  MoveL 1331 to (-194.97, 429.6, -4.48) mm, rotated rx -180 ry 0 rz -11.91 deg; joints [13.946, -29.664, 81.646, -88.075, 90.999, 141.138]
  MoveL 1332 to (-195.21, 429.6, -4.47) mm, rotated rx -180 ry 0 rz -11.91 deg; joints [13.938, -29.668, 81.653, -88.081, 90.994, 141.141]
  MoveL 1333 to (-195.45, 429.58, -4.47) mm, rotated rx -180 ry 0 rz -11.91 deg; joints [13.931, -29.672, 81.662, -88.087, 90.989, 141.146]
  MoveL 1334 to (-195.69, 429.55, -4.48) mm, rotated rx -180 ry 0 rz -11.91 deg; joints [13.923, -29.676, 81.673, -88.093, 90.984, 141.152]
  MoveL 1335 to (-195.93, 429.49, -4.47) mm, rotated rx -180 ry 0 rz -11.91 deg; joints [13.916, -29.682, 81.686, -88.098, 90.979, 141.159]
  MoveL 1336 to (-196.18, 429.42, -4.47) mm, rotated rx -180 ry 0 rz -11.91 deg; joints [13.909, -29.689, 81.701, -88.104, 90.974, 141.167]
  MoveL 1337 to (-196.42, 429.32, -4.47) mm, rotated rx -180 ry 0 rz -11.91 deg; joints [13.902, -29.698, 81.719, -88.109, 90.97, 141.176]
  MoveL 1338 to (-196.6, 429.23, -4.48) mm, rotated rx -180 ry 0 rz -11.91 deg; joints [13.896, -29.704, 81.734, -88.113, 90.966, 141.184]
  MoveL 1339 to (-196.78, 429.13, -4.47) mm, rotated rx -180 ry 0 rz -11.91 deg; joints [13.891, -29.712, 81.751, -88.117, 90.963, 141.193]
  MoveL 1340 to (-196.95, 429, -4.48) mm, rotated rx -180 ry 0 rz -11.91 deg; joints [13.887, -29.721, 81.769, -88.121, 90.96, 141.203]
  MoveL 1341 to (-197.13, 428.87, -4.48) mm, rotated rx -180 ry 0 rz -11.91 deg; joints [13.882, -29.73, 81.79, -88.124, 90.956, 141.214]
  MoveL 1342 to (-197.37, 428.65, -4.47) mm, rotated rx -180 ry 0 rz -11.91 deg; joints [13.876, -29.744, 81.82, -88.128, 90.952, 141.231]
  MoveL 1343 to (-197.56, 428.44, -4.47) mm, rotated rx -180 ry 0 rz -11.91 deg; joints [13.872, -29.758, 81.85, -88.132, 90.949, 141.246]
  MoveL 1344 to (-197.72, 428.22, -4.48) mm, rotated rx 180 ry 0 rz -11.91 deg; joints [13.868, -29.771, 81.878, -88.134, 90.946, 141.262]
  MoveL 1345 to (-197.85, 428.01, -4.48) mm, rotated rx 180 ry 0 rz -11.91 deg; joints [13.865, -29.783, 81.906, -88.136, 90.944, 141.277]
  MoveL 1346 to (-197.98, 427.77, -4.47) mm, rotated rx -180 ry 0 rz -11.91 deg; joints [13.863, -29.797, 81.937, -88.137, 90.942, 141.293]
  MoveL 1347 to (-198.08, 427.53, -4.48) mm, rotated rx -180 ry 0 rz -11.91 deg; joints [13.862, -29.811, 81.966, -88.138, 90.941, 141.309]
  MoveL 1348 to (-198.16, 427.29, -4.48) mm, rotated rx -180 ry 0 rz -11.91 deg; joints [13.861, -29.825, 81.996, -88.138, 90.94, 141.325]
  MoveL 1349 to (-198.21, 427.04, -4.48) mm, rotated rx -180 ry 0 rz -11.91 deg; joints [13.861, -29.838, 82.024, -88.138, 90.94, 141.34]
  MoveL 1350 to (-198.25, 426.8, -4.48) mm, rotated rx -180 ry 0 rz -11.91 deg; joints [13.862, -29.851, 82.053, -88.137, 90.94, 141.356]
  MoveL 1351 to (-198.27, 426.56, -4.48) mm, rotated rx 180 ry 0 rz -11.91 deg; joints [13.864, -29.864, 82.08, -88.136, 90.94, 141.37]
  MoveL 1352 to (-198.27, 426.08, -4.48) mm, rotated rx 180 ry 0 rz -11.91 deg; joints [13.867, -29.889, 82.134, -88.133, 90.941, 141.4]
  MoveL 1353 to (-198.27, 425.59, -4.48) mm, rotated rx -180 ry 0 rz -11.91 deg; joints [13.871, -29.914, 82.188, -88.129, 90.943, 141.429]
  MoveL 1354 to (-198.25, 425.35, -4.47) mm, rotated rx -180 ry 0 rz -11.91 deg; joints [13.874, -29.926, 82.215, -88.127, 90.944, 141.443]
  MoveL 1355 to (-198.22, 425.11, -4.47) mm, rotated rx -180 ry 0 rz -11.91 deg; joints [13.877, -29.938, 82.241, -88.124, 90.945, 141.457]
  MoveL 1356 to (-198.16, 424.87, -4.48) mm, rotated rx -180 ry 0 rz -11.91 deg; joints [13.881, -29.95, 82.266, -88.121, 90.947, 141.471]
  MoveL 1357 to (-198.09, 424.63, -4.48) mm, rotated rx -180 ry 0 rz -11.91 deg; joints [13.885, -29.961, 82.291, -88.117, 90.949, 141.484]
  MoveL 1358 to (-197.99, 424.39, -4.48) mm, rotated rx -180 ry 0 rz -11.91 deg; joints [13.89, -29.972, 82.315, -88.113, 90.952, 141.498]
  MoveL 1359 to (-197.87, 424.15, -4.47) mm, rotated rx -180 ry 0 rz -11.91 deg; joints [13.896, -29.983, 82.339, -88.108, 90.955, 141.51]
  MoveL 1360 to (-197.73, 423.93, -4.48) mm, rotated rx 180 ry 0 rz -11.91 deg; joints [13.902, -29.993, 82.36, -88.103, 90.959, 141.522]
  MoveL 1361 to (-197.57, 423.71, -4.47) mm, rotated rx -180 ry 0 rz -11.91 deg; joints [13.91, -30.002, 82.38, -88.097, 90.963, 141.532]
  MoveL 1362 to (-197.38, 423.49, -4.48) mm, rotated rx 180 ry 0 rz -11.91 deg; joints [13.918, -30.011, 82.399, -88.09, 90.967, 141.543]
  MoveL 1363 to (-197.14, 423.27, -4.47) mm, rotated rx -180 ry 0 rz -11.91 deg; joints [13.927, -30.019, 82.417, -88.083, 90.973, 141.553]
  MoveL 1364 to (-196.96, 423.13, -4.47) mm, rotated rx -180 ry 0 rz -11.91 deg; joints [13.934, -30.025, 82.428, -88.077, 90.977, 141.558]
  MoveL 1365 to (-196.78, 423, -4.48) mm, rotated rx 180 ry 0 rz -11.91 deg; joints [13.941, -30.029, 82.436, -88.071, 90.981, 141.563]
  MoveL 1366 to (-196.6, 422.9, -4.48) mm, rotated rx -180 ry 0 rz -11.91 deg; joints [13.948, -30.032, 82.443, -88.066, 90.985, 141.567]
  MoveL 1367 to (-196.42, 422.81, -4.48) mm, rotated rx 180 ry 0 rz -11.91 deg; joints [13.955, -30.034, 82.448, -88.061, 90.989, 141.57]
  MoveL 1368 to (-196.18, 422.71, -4.48) mm, rotated rx -180 ry 0 rz -11.91 deg; joints [13.963, -30.036, 82.452, -88.054, 90.994, 141.572]
  MoveL 1369 to (-195.93, 422.63, -4.48) mm, rotated rx 180 ry 0 rz -11.91 deg; joints [13.972, -30.037, 82.454, -88.047, 90.999, 141.573]
  MoveL 1370 to (-195.69, 422.58, -4.48) mm, rotated rx 180 ry 0 rz -11.91 deg; joints [13.98, -30.037, 82.453, -88.04, 91.004, 141.573]
  MoveL 1371 to (-195.45, 422.54, -4.47) mm, rotated rx -180 ry 0 rz -11.91 deg; joints [13.988, -30.036, 82.451, -88.034, 91.01, 141.572]
  MoveL 1372 to (-195.21, 422.52, -4.48) mm, rotated rx -180 ry 0 rz -11.91 deg; joints [13.996, -30.034, 82.446, -88.028, 91.015, 141.569]
  MoveL 1373 to (-194.97, 422.52, -4.47) mm, rotated rx -180 ry 0 rz -11.91 deg; joints [14.004, -30.031, 82.439, -88.021, 91.019, 141.566]
  Set speed (38.1 mm/s)
  MoveL 1374 to (-194.97, 421.25, -4.48) mm, rotated rx -180 ry 0 rz -11.91 deg; joints [14.015, -30.096, 82.581, -88.012, 91.023, 141.642]
  MoveL 1375 to (-195.61, 421.25, -4.48) mm, rotated rx -180 ry 0 rz -11.91 deg; joints [13.994, -30.104, 82.599, -88.028, 91.01, 141.651]
  Set speed (25.4 mm/s)
  MoveL 1376 to (-195.61, 421.25, -6.84) mm, rotated rx -180 ry 0 rz -11.91 deg; joints [13.994, -29.993, 82.575, -88.026, 91.008, 141.739]
  MoveL 1377 to (-195.61, 421.89, -7.47) mm, rotated rx -180 ry 0 rz -11.91 deg; joints [13.989, -29.93, 82.498, -88.03, 91.005, 141.724]
  Set speed (38.1 mm/s)
  MoveL 1378 to (-194.97, 422.52, -7.47) mm, rotated rx 180 ry 0 rz -11.91 deg; joints [14.005, -29.89, 82.41, -88.019, 91.016, 141.677]
  Set speed (76.2 mm/s)
  MoveL 1379 to (213.41, 422.52, -7.48) mm, rotated rx -180 ry 0 rz -11.91 deg; joints [26.411, -21.408, 63.956, -79.718, 100.425, 132.671]
  MoveL 1380 to (213.89, 422.53, -7.47) mm, rotated rx -180 ry 0 rz -11.91 deg; joints [26.425, -21.393, 63.923, -79.712, 100.438, 132.655]
  MoveL 1381 to (214.13, 422.55, -7.48) mm, rotated rx -180 ry 0 rz -11.91 deg; joints [26.431, -21.384, 63.904, -79.71, 100.445, 132.646]
  MoveL 1382 to (214.37, 422.59, -7.48) mm, rotated rx 180 ry 0 rz -11.91 deg; joints [26.437, -21.374, 63.882, -79.707, 100.451, 132.635]
  MoveL 1383 to (214.61, 422.65, -7.48) mm, rotated rx -180 ry 0 rz -11.91 deg; joints [26.443, -21.362, 63.858, -79.706, 100.458, 132.623]
  MoveL 1384 to (214.85, 422.74, -7.47) mm, rotated rx 180 ry 0 rz -11.91 deg; joints [26.449, -21.35, 63.831, -79.704, 100.464, 132.609]
  MoveL 1385 to (215.09, 422.84, -7.47) mm, rotated rx -180 ry 0 rz -11.91 deg; joints [26.454, -21.335, 63.801, -79.704, 100.471, 132.594]
  MoveL 1386 to (215.34, 422.97, -7.48) mm, rotated rx -180 ry 0 rz -11.91 deg; joints [26.459, -21.319, 63.767, -79.703, 100.478, 132.577]
  MoveL 1387 to (215.58, 423.13, -7.47) mm, rotated rx -180 ry 0 rz -11.91 deg; joints [26.463, -21.302, 63.729, -79.704, 100.484, 132.558]
  MoveL 1388 to (215.82, 423.33, -7.47) mm, rotated rx 180 ry 0 rz -11.91 deg; joints [26.467, -21.282, 63.687, -79.705, 100.491, 132.536]
  MoveL 1389 to (215.96, 423.46, -7.48) mm, rotated rx 180 ry 0 rz -11.91 deg; joints [26.469, -21.268, 63.659, -79.706, 100.495, 132.521]
  MoveL 1390 to (216.09, 423.6, -7.48) mm, rotated rx 180 ry 0 rz -11.91 deg; joints [26.471, -21.256, 63.632, -79.708, 100.499, 132.508]
  MoveL 1391 to (216.2, 423.73, -7.48) mm, rotated rx -180 ry 0 rz -11.91 deg; joints [26.472, -21.244, 63.607, -79.71, 100.502, 132.494]
  MoveL 1392 to (216.3, 423.87, -7.48) mm, rotated rx -180 ry 0 rz -11.91 deg; joints [26.473, -21.232, 63.582, -79.711, 100.505, 132.481]
  MoveL 1393 to (216.39, 424.01, -7.48) mm, rotated rx -180 ry 0 rz -11.91 deg; joints [26.474, -21.22, 63.557, -79.713, 100.508, 132.468]
  MoveL 1394 to (216.47, 424.15, -7.48) mm, rotated rx -180 ry 0 rz -11.91 deg; joints [26.474, -21.209, 63.532, -79.715, 100.511, 132.455]
  MoveL 1395 to (216.6, 424.39, -7.48) mm, rotated rx -180 ry 0 rz -11.91 deg; joints [26.474, -21.189, 63.492, -79.719, 100.515, 132.434]
  MoveL 1396 to (216.69, 424.63, -7.48) mm, rotated rx -180 ry 0 rz -11.91 deg; joints [26.474, -21.171, 63.452, -79.723, 100.518, 132.413]
  MoveL 1397 to (216.77, 424.87, -7.47) mm, rotated rx -180 ry 0 rz -11.91 deg; joints [26.472, -21.153, 63.415, -79.728, 100.521, 132.393]
  MoveL 1398 to (216.82, 425.11, -7.48) mm, rotated rx 180 ry 0 rz -11.91 deg; joints [26.47, -21.135, 63.378, -79.733, 100.523, 132.374]
  MoveL 1399 to (216.86, 425.35, -7.48) mm, rotated rx -180 ry 0 rz -11.91 deg; joints [26.468, -21.119, 63.343, -79.738, 100.524, 132.355]
  MoveL 1400 to (216.88, 425.59, -7.47) mm, rotated rx -180 ry 0 rz -11.91 deg; joints [26.465, -21.103, 63.309, -79.743, 100.525, 132.337]
  MoveL 1401 to (216.88, 426.08, -7.48) mm, rotated rx -180 ry 0 rz -11.91 deg; joints [26.459, -21.071, 63.244, -79.754, 100.527, 132.301]
  MoveL 1402 to (216.88, 427.04, -7.47) mm, rotated rx -180 ry 0 rz -11.91 deg; joints [26.445, -21.009, 63.112, -79.776, 100.529, 132.231]
  MoveL 1403 to (216.86, 427.29, -7.47) mm, rotated rx 180 ry 0 rz -11.91 deg; joints [26.441, -20.994, 63.08, -79.781, 100.529, 132.213]
  MoveL 1404 to (216.83, 427.53, -7.47) mm, rotated rx -180 ry 0 rz -11.91 deg; joints [26.437, -20.979, 63.05, -79.787, 100.529, 132.197]
  MoveL 1405 to (216.78, 427.77, -7.48) mm, rotated rx 180 ry 0 rz -11.91 deg; joints [26.432, -20.965, 63.02, -79.793, 100.528, 132.181]
  MoveL 1406 to (216.71, 428.01, -7.47) mm, rotated rx -180 ry 0 rz -11.91 deg; joints [26.427, -20.952, 62.992, -79.8, 100.527, 132.165]
  MoveL 1407 to (216.63, 428.21, -7.48) mm, rotated rx -180 ry 0 rz -11.91 deg; joints [26.422, -20.942, 62.97, -79.805, 100.525, 132.153]
  MoveL 1408 to (216.54, 428.41, -7.47) mm, rotated rx -180 ry 0 rz -11.91 deg; joints [26.417, -20.932, 62.949, -79.811, 100.523, 132.141]
  MoveL 1409 to (216.43, 428.61, -7.48) mm, rotated rx -180 ry 0 rz -11.91 deg; joints [26.411, -20.922, 62.93, -79.817, 100.521, 132.13]
  MoveL 1410 to (216.3, 428.81, -7.48) mm, rotated rx 180 ry 0 rz -11.91 deg; joints [26.405, -20.913, 62.911, -79.823, 100.518, 132.12]
  MoveL 1411 to (216.16, 428.99, -7.48) mm, rotated rx 180 ry 0 rz -11.91 deg; joints [26.398, -20.906, 62.896, -79.829, 100.515, 132.111]
  MoveL 1412 to (215.99, 429.18, -7.48) mm, rotated rx -180 ry 0 rz -11.91 deg; joints [26.391, -20.899, 62.882, -79.835, 100.511, 132.103]
  MoveL 1413 to (215.78, 429.38, -7.48) mm, rotated rx -180 ry 0 rz -11.91 deg; joints [26.383, -20.893, 62.868, -79.843, 100.506, 132.095]
  MoveL 1414 to (215.57, 429.55, -7.48) mm, rotated rx -180 ry 0 rz -11.91 deg; joints [26.374, -20.889, 62.86, -79.849, 100.501, 132.089]
  MoveL 1415 to (215.39, 429.67, -7.48) mm, rotated rx -180 ry 0 rz -11.91 deg; joints [26.368, -20.886, 62.855, -79.854, 100.496, 132.086]
  MoveL 1416 to (215.21, 429.78, -7.48) mm, rotated rx -180 ry 0 rz -11.91 deg; joints [26.361, -20.885, 62.853, -79.859, 100.491, 132.084]
  MoveL 1417 to (215.02, 429.87, -7.48) mm, rotated rx -180 ry 0 rz -11.91 deg; joints [26.355, -20.885, 62.853, -79.863, 100.487, 132.083]
  MoveL 1418 to (214.84, 429.94, -7.48) mm, rotated rx -180 ry 0 rz -11.91 deg; joints [26.349, -20.886, 62.855, -79.867, 100.482, 132.084]
  MoveL 1419 to (214.61, 430.02, -7.47) mm, rotated rx 180 ry 0 rz -11.91 deg; joints [26.341, -20.888, 62.86, -79.872, 100.476, 132.085]
  MoveL 1420 to (214.37, 430.08, -7.48) mm, rotated rx 180 ry 0 rz -11.91 deg; joints [26.334, -20.892, 62.868, -79.876, 100.47, 132.088]
  MoveL 1421 to (214.13, 430.13, -7.48) mm, rotated rx 180 ry 0 rz -11.91 deg; joints [26.326, -20.897, 62.879, -79.88, 100.464, 132.093]
  MoveL 1422 to (213.89, 430.15, -7.48) mm, rotated rx -180 ry 0 rz -11.91 deg; joints [26.319, -20.903, 62.892, -79.884, 100.457, 132.099]
  MoveL 1423 to (213.41, 430.15, -7.48) mm, rotated rx 180 ry 0 rz -11.91 deg; joints [26.306, -20.918, 62.924, -79.89, 100.444, 132.114]
  MoveL 1424 to (-194.49, 430.15, -7.48) mm, rotated rx 180 ry 0 rz -11.91 deg; joints [13.958, -29.49, 81.541, -88.064, 91.004, 141.207]
  MoveL 1425 to (-195.36, 430.14, -7.48) mm, rotated rx -180 ry 0 rz -11.91 deg; joints [13.93, -29.501, 81.567, -88.086, 90.986, 141.221]
  MoveL 1426 to (-195.58, 430.12, -7.48) mm, rotated rx 180 ry 0 rz -11.91 deg; joints [13.923, -29.505, 81.576, -88.091, 90.981, 141.226]
  MoveL 1427 to (-195.8, 430.08, -7.47) mm, rotated rx 180 ry 0 rz -11.91 deg; joints [13.916, -29.51, 81.587, -88.097, 90.977, 141.232]
  MoveL 1428 to (-196.02, 430.02, -7.48) mm, rotated rx 180 ry 0 rz -11.91 deg; joints [13.91, -29.516, 81.599, -88.102, 90.973, 141.238]
  MoveL 1429 to (-196.24, 429.94, -7.48) mm, rotated rx 180 ry 0 rz -11.91 deg; joints [13.903, -29.523, 81.614, -88.107, 90.968, 141.246]
  MoveL 1430 to (-196.42, 429.87, -7.48) mm, rotated rx 180 ry 0 rz -11.91 deg; joints [13.898, -29.529, 81.627, -88.111, 90.965, 141.253]
  MoveL 1431 to (-196.56, 429.8, -7.47) mm, rotated rx -180 ry 0 rz -11.91 deg; joints [13.894, -29.534, 81.64, -88.114, 90.962, 141.26]
  MoveL 1432 to (-196.71, 429.71, -7.48) mm, rotated rx -180 ry 0 rz -11.91 deg; joints [13.89, -29.54, 81.653, -88.117, 90.959, 141.267]
  MoveL 1433 to (-196.86, 429.62, -7.47) mm, rotated rx -180 ry 0 rz -11.91 deg; joints [13.885, -29.547, 81.667, -88.12, 90.957, 141.275]
  MoveL 1434 to (-197.01, 429.52, -7.47) mm, rotated rx 180 ry 0 rz -11.91 deg; joints [13.882, -29.554, 81.683, -88.123, 90.954, 141.283]
  MoveL 1435 to (-197.15, 429.4, -7.47) mm, rotated rx -180 ry 0 rz -11.91 deg; joints [13.878, -29.562, 81.701, -88.126, 90.951, 141.293]
  MoveL 1436 to (-197.3, 429.27, -7.47) mm, rotated rx 180 ry 0 rz -11.91 deg; joints [13.874, -29.571, 81.72, -88.129, 90.949, 141.303]
  MoveL 1437 to (-197.46, 429.1, -7.48) mm, rotated rx -180 ry 0 rz -11.91 deg; joints [13.87, -29.582, 81.742, -88.132, 90.946, 141.315]
  MoveL 1438 to (-197.6, 428.94, -7.48) mm, rotated rx 180 ry 0 rz -11.91 deg; joints [13.867, -29.592, 81.765, -88.134, 90.943, 141.327]
  MoveL 1439 to (-197.76, 428.71, -7.48) mm, rotated rx -180 ry 0 rz -11.91 deg; joints [13.863, -29.606, 81.795, -88.137, 90.941, 141.344]
  MoveL 1440 to (-197.9, 428.47, -7.47) mm, rotated rx 180 ry 0 rz -11.91 deg; joints [13.861, -29.62, 81.825, -88.138, 90.939, 141.36]
  MoveL 1441 to (-198.01, 428.24, -7.48) mm, rotated rx -180 ry 0 rz -11.91 deg; joints [13.859, -29.633, 81.854, -88.139, 90.937, 141.375]
  MoveL 1442 to (-198.1, 428.01, -7.48) mm, rotated rx -180 ry 0 rz -11.91 deg; joints [13.858, -29.646, 81.883, -88.14, 90.936, 141.391]
  MoveL 1443 to (-198.17, 427.77, -7.48) mm, rotated rx -180 ry 0 rz -11.91 deg; joints [13.858, -29.659, 81.912, -88.14, 90.935, 141.406]
  MoveL 1444 to (-198.23, 427.53, -7.47) mm, rotated rx -180 ry 0 rz -11.91 deg; joints [13.858, -29.673, 81.941, -88.14, 90.935, 141.422]
  MoveL 1445 to (-198.26, 427.29, -7.47) mm, rotated rx -180 ry 0 rz -11.91 deg; joints [13.859, -29.686, 81.969, -88.139, 90.935, 141.437]
  MoveL 1446 to (-198.27, 427.04, -7.48) mm, rotated rx -180 ry 0 rz -11.91 deg; joints [13.86, -29.698, 81.996, -88.137, 90.935, 141.452]
  MoveL 1447 to (-198.27, 426.08, -7.47) mm, rotated rx 180 ry 0 rz -11.91 deg; joints [13.868, -29.748, 82.104, -88.13, 90.938, 141.51]
  MoveL 1448 to (-198.27, 425.59, -7.48) mm, rotated rx -180 ry 0 rz -11.91 deg; joints [13.872, -29.773, 82.158, -88.126, 90.94, 141.539]
  MoveL 1449 to (-198.25, 425.35, -7.47) mm, rotated rx -180 ry 0 rz -11.91 deg; joints [13.875, -29.785, 82.185, -88.124, 90.941, 141.554]
  MoveL 1450 to (-198.22, 425.11, -7.48) mm, rotated rx -180 ry 0 rz -11.91 deg; joints [13.878, -29.797, 82.211, -88.122, 90.942, 141.568]
  MoveL 1451 to (-198.16, 424.87, -7.48) mm, rotated rx -180 ry 0 rz -11.91 deg; joints [13.881, -29.809, 82.236, -88.118, 90.944, 141.582]
  MoveL 1452 to (-198.09, 424.63, -7.48) mm, rotated rx -180 ry 0 rz -11.91 deg; joints [13.886, -29.821, 82.261, -88.115, 90.946, 141.595]
  MoveL 1453 to (-197.99, 424.39, -7.48) mm, rotated rx -180 ry 0 rz -11.91 deg; joints [13.891, -29.832, 82.286, -88.11, 90.949, 141.608]
  MoveL 1454 to (-197.87, 424.15, -7.47) mm, rotated rx -180 ry 0 rz -11.91 deg; joints [13.897, -29.843, 82.309, -88.105, 90.952, 141.621]
  MoveL 1455 to (-197.73, 423.93, -7.48) mm, rotated rx -180 ry 0 rz -11.91 deg; joints [13.903, -29.852, 82.33, -88.1, 90.956, 141.632]
  MoveL 1456 to (-197.57, 423.71, -7.48) mm, rotated rx 180 ry 0 rz -11.91 deg; joints [13.91, -29.862, 82.35, -88.094, 90.96, 141.643]
  MoveL 1457 to (-197.38, 423.49, -7.48) mm, rotated rx 180 ry 0 rz -11.91 deg; joints [13.918, -29.87, 82.369, -88.088, 90.964, 141.654]
  MoveL 1458 to (-197.14, 423.27, -7.48) mm, rotated rx 180 ry 0 rz -11.91 deg; joints [13.928, -29.879, 82.387, -88.08, 90.97, 141.663]
  MoveL 1459 to (-196.96, 423.13, -7.48) mm, rotated rx 180 ry 0 rz -11.91 deg; joints [13.935, -29.884, 82.398, -88.074, 90.974, 141.669]
  MoveL 1460 to (-196.78, 423, -7.48) mm, rotated rx -180 ry 0 rz -11.91 deg; joints [13.942, -29.888, 82.406, -88.069, 90.978, 141.674]
  MoveL 1461 to (-196.6, 422.9, -7.47) mm, rotated rx -180 ry 0 rz -11.91 deg; joints [13.949, -29.891, 82.413, -88.063, 90.982, 141.678]
  MoveL 1462 to (-196.42, 422.81, -7.48) mm, rotated rx 180 ry 0 rz -11.91 deg; joints [13.955, -29.893, 82.418, -88.058, 90.986, 141.68]
  MoveL 1463 to (-196.18, 422.71, -7.48) mm, rotated rx -180 ry 0 rz -11.91 deg; joints [13.964, -29.895, 82.422, -88.051, 90.991, 141.683]
  MoveL 1464 to (-195.93, 422.63, -7.47) mm, rotated rx -180 ry 0 rz -11.91 deg; joints [13.973, -29.896, 82.424, -88.044, 90.996, 141.684]
  MoveL 1465 to (-195.69, 422.58, -7.48) mm, rotated rx -180 ry 0 rz -11.91 deg; joints [13.981, -29.896, 82.423, -88.038, 91.001, 141.684]
  MoveL 1466 to (-195.45, 422.54, -7.47) mm, rotated rx 180 ry 0 rz -11.91 deg; joints [13.989, -29.895, 82.421, -88.031, 91.006, 141.682]
  MoveL 1467 to (-195.21, 422.52, -7.47) mm, rotated rx 180 ry 0 rz -11.91 deg; joints [13.997, -29.893, 82.416, -88.025, 91.011, 141.68]
  MoveL 1468 to (-194.97, 422.52, -7.47) mm, rotated rx 180 ry 0 rz -11.91 deg; joints [14.005, -29.89, 82.41, -88.019, 91.016, 141.677]
  Set speed (38.1 mm/s)
  MoveL 1469 to (-194.97, 421.25, -7.48) mm, rotated rx -180 ry 0 rz -11.91 deg; joints [14.015, -29.955, 82.551, -88.009, 91.02, 141.753]
  MoveL 1470 to (-195.61, 421.25, -7.47) mm, rotated rx 180 ry 0 rz -11.91 deg; joints [13.995, -29.963, 82.569, -88.026, 91.007, 141.762]
  Set speed (25.4 mm/s)
  MoveL 1471 to (-195.61, 421.25, -9.84) mm, rotated rx -180 ry 0 rz -11.91 deg; joints [13.995, -29.852, 82.545, -88.023, 91.004, 141.85]
  MoveL 1472 to (-195.61, 421.89, -10.48) mm, rotated rx 180 ry 0 rz -11.91 deg; joints [13.99, -29.789, 82.467, -88.028, 91.002, 141.835]
  Set speed (38.1 mm/s)
  MoveL 1473 to (-194.97, 422.52, -10.48) mm, rotated rx -180 ry 0 rz -11.91 deg; joints [14.006, -29.749, 82.379, -88.016, 91.013, 141.787]
  Set speed (76.2 mm/s)
  MoveL 1474 to (213.41, 422.52, -10.48) mm, rotated rx -180 ry 0 rz -11.91 deg; joints [26.412, -21.277, 63.92, -79.7, 100.409, 132.767]
  MoveL 1475 to (213.89, 422.53, -10.48) mm, rotated rx -180 ry 0 rz -11.91 deg; joints [26.426, -21.261, 63.887, -79.694, 100.422, 132.751]
  MoveL 1476 to (214.13, 422.55, -10.48) mm, rotated rx -180 ry 0 rz -11.91 deg; joints [26.432, -21.252, 63.868, -79.692, 100.428, 132.742]
  MoveL 1477 to (214.37, 422.59, -10.48) mm, rotated rx -180 ry 0 rz -11.91 deg; joints [26.438, -21.242, 63.846, -79.689, 100.435, 132.731]
  MoveL 1478 to (214.61, 422.65, -10.48) mm, rotated rx -180 ry 0 rz -11.91 deg; joints [26.444, -21.23, 63.822, -79.688, 100.441, 132.719]
  MoveL 1479 to (214.85, 422.74, -10.47) mm, rotated rx 180 ry 0 rz -11.91 deg; joints [26.45, -21.218, 63.795, -79.686, 100.448, 132.705]
  MoveL 1480 to (215.09, 422.84, -10.47) mm, rotated rx 180 ry 0 rz -11.91 deg; joints [26.455, -21.203, 63.764, -79.686, 100.454, 132.69]
  MoveL 1481 to (215.34, 422.97, -10.48) mm, rotated rx -180 ry 0 rz -11.91 deg; joints [26.46, -21.187, 63.731, -79.685, 100.461, 132.673]
  MoveL 1482 to (215.58, 423.13, -10.47) mm, rotated rx 180 ry 0 rz -11.91 deg; joints [26.464, -21.17, 63.693, -79.686, 100.468, 132.654]
  MoveL 1483 to (215.82, 423.33, -10.48) mm, rotated rx -180 ry 0 rz -11.91 deg; joints [26.468, -21.15, 63.651, -79.687, 100.475, 132.632]
  MoveL 1484 to (215.96, 423.46, -10.48) mm, rotated rx 180 ry 0 rz -11.91 deg; joints [26.47, -21.137, 63.623, -79.688, 100.479, 132.617]
  MoveL 1485 to (216.09, 423.6, -10.48) mm, rotated rx -180 ry 0 rz -11.91 deg; joints [26.472, -21.124, 63.596, -79.69, 100.483, 132.604]
  MoveL 1486 to (216.2, 423.73, -10.48) mm, rotated rx -180 ry 0 rz -11.91 deg; joints [26.473, -21.112, 63.57, -79.691, 100.486, 132.59]
  MoveL 1487 to (216.3, 423.87, -10.47) mm, rotated rx -180 ry 0 rz -11.91 deg; joints [26.474, -21.1, 63.545, -79.693, 100.489, 132.577]
  MoveL 1488 to (216.39, 424.01, -10.47) mm, rotated rx -180 ry 0 rz -11.91 deg; joints [26.475, -21.088, 63.52, -79.695, 100.492, 132.564]
  MoveL 1489 to (216.47, 424.15, -10.47) mm, rotated rx -180 ry 0 rz -11.91 deg; joints [26.475, -21.077, 63.496, -79.697, 100.494, 132.551]
  MoveL 1490 to (216.69, 424.27, -10.48) mm, rotated rx 180 ry 0 rz -11.91 deg; joints [26.479, -21.062, 63.465, -79.697, 100.501, 132.535]
  MoveL 1491 to (219.83, 424.27, -10.48) mm, rotated rx -180 ry 0 rz -11.91 deg; joints [26.566, -20.963, 63.253, -79.657, 100.584, 132.434]
  MoveL 1492 to (220.05, 424.15, -10.48) mm, rotated rx -180 ry 0 rz -11.91 deg; joints [26.574, -20.963, 63.254, -79.651, 100.59, 132.436]
  MoveL 1493 to (220.05, 53.41, -10.47) mm, rotated rx -180 ry 0 rz -11.91 deg; joints [32.834, -38.199, 100.656, -71.009, 99.189, 153.203]
  MoveL 1494 to (219.83, 53.17, -10.47) mm, rotated rx -180 ry 0 rz -11.91 deg; joints [32.832, -38.213, 100.687, -71.008, 99.182, 153.219]
  MoveL 1495 to (-199.12, 53.17, -10.48) mm, rotated rx -180 ry 0 rz -11.91 deg; joints [17.67, -44.811, 116.798, -84.307, 91.428, 161.21]
  MoveL 1496 to (-199.7, 53.17, -10.48) mm, rotated rx -180 ry 0 rz -11.91 deg; joints [17.647, -44.817, 116.813, -84.329, 91.42, 161.218]
  MoveL 1497 to (-199.9, 53.41, -10.48) mm, rotated rx -180 ry 0 rz -11.91 deg; joints [17.636, -44.811, 116.799, -84.339, 91.418, 161.21]
  MoveL 1498 to (-199.9, 424.15, -10.47) mm, rotated rx -180 ry 0 rz -11.91 deg; joints [13.831, -29.727, 82.335, -88.155, 90.908, 141.761]
  MoveL 1499 to (-199.7, 424.27, -10.48) mm, rotated rx -180 ry 0 rz -11.91 deg; joints [13.837, -29.718, 82.316, -88.151, 90.911, 141.751]
  MoveL 1500 to (-198.11, 424.27, -10.47) mm, rotated rx -180 ry 0 rz -11.91 deg; joints [13.889, -29.698, 82.272, -88.11, 90.944, 141.728]
  MoveL 1501 to (-197.87, 424.15, -10.47) mm, rotated rx -180 ry 0 rz -11.91 deg; joints [13.898, -29.702, 82.278, -88.103, 90.949, 141.731]
  MoveL 1502 to (-197.73, 423.93, -10.47) mm, rotated rx -180 ry 0 rz -11.91 deg; joints [13.904, -29.711, 82.299, -88.098, 90.952, 141.743]
  MoveL 1503 to (-197.57, 423.71, -10.47) mm, rotated rx 180 ry 0 rz -11.91 deg; joints [13.911, -29.72, 82.319, -88.092, 90.956, 141.754]
  MoveL 1504 to (-197.38, 423.49, -10.48) mm, rotated rx -180 ry 0 rz -11.91 deg; joints [13.919, -29.729, 82.338, -88.085, 90.961, 141.764]
  MoveL 1505 to (-197.14, 423.27, -10.48) mm, rotated rx -180 ry 0 rz -11.91 deg; joints [13.929, -29.738, 82.356, -88.078, 90.966, 141.774]
  MoveL 1506 to (-196.96, 423.13, -10.47) mm, rotated rx 180 ry 0 rz -11.91 deg; joints [13.936, -29.743, 82.367, -88.072, 90.97, 141.78]
  MoveL 1507 to (-196.78, 423, -10.48) mm, rotated rx -180 ry 0 rz -11.91 deg; joints [13.943, -29.747, 82.376, -88.066, 90.975, 141.784]
  MoveL 1508 to (-196.6, 422.9, -10.48) mm, rotated rx -180 ry 0 rz -11.91 deg; joints [13.949, -29.75, 82.382, -88.061, 90.979, 141.788]
  MoveL 1509 to (-196.42, 422.81, -10.48) mm, rotated rx -180 ry 0 rz -11.91 deg; joints [13.956, -29.752, 82.387, -88.056, 90.982, 141.791]
  MoveL 1510 to (-196.18, 422.71, -10.48) mm, rotated rx 180 ry 0 rz -11.91 deg; joints [13.965, -29.754, 82.392, -88.049, 90.988, 141.793]
  MoveL 1511 to (-195.93, 422.63, -10.48) mm, rotated rx -180 ry 0 rz -11.91 deg; joints [13.973, -29.755, 82.393, -88.042, 90.993, 141.794]
  MoveL 1512 to (-195.69, 422.58, -10.48) mm, rotated rx -180 ry 0 rz -11.91 deg; joints [13.982, -29.755, 82.393, -88.035, 90.998, 141.794]
  MoveL 1513 to (-195.45, 422.54, -10.48) mm, rotated rx -180 ry 0 rz -11.91 deg; joints [13.99, -29.754, 82.39, -88.029, 91.003, 141.793]
  MoveL 1514 to (-195.21, 422.52, -10.47) mm, rotated rx 180 ry 0 rz -11.91 deg; joints [13.998, -29.752, 82.385, -88.022, 91.008, 141.79]
  MoveL 1515 to (-194.97, 422.52, -10.48) mm, rotated rx -180 ry 0 rz -11.91 deg; joints [14.006, -29.749, 82.379, -88.016, 91.013, 141.787]
  Set speed (38.1 mm/s)
  MoveL 1516 to (-194.97, 421.25, -10.48) mm, rotated rx -180 ry 0 rz -11.91 deg; joints [14.016, -29.814, 82.52, -88.007, 91.016, 141.864]
  MoveL 1517 to (-195.61, 421.25, -10.47) mm, rotated rx -180 ry 0 rz -11.91 deg; joints [13.995, -29.822, 82.538, -88.023, 91.003, 141.873]
  Set speed (25.4 mm/s)
  MoveL 1518 to (-195.61, 421.25, -12.84) mm, rotated rx 180 ry 0 rz -11.91 deg; joints [13.996, -29.71, 82.513, -88.021, 91.001, 141.96]
  MoveL 1519 to (-195.61, 421.89, -13.48) mm, rotated rx -180 ry 0 rz -11.91 deg; joints [13.991, -29.648, 82.436, -88.025, 90.998, 141.945]
  Set speed (38.1 mm/s)
  MoveL 1520 to (-194.97, 422.52, -13.48) mm, rotated rx 180 ry 0 rz -11.91 deg; joints [14.006, -29.607, 82.348, -88.014, 91.009, 141.897]
  Set speed (76.2 mm/s)
  MoveL 1521 to (213.41, 422.52, -13.48) mm, rotated rx -180 ry 0 rz -11.91 deg; joints [26.413, -21.144, 63.884, -79.682, 100.392, 132.863]
  MoveL 1522 to (213.89, 422.53, -13.47) mm, rotated rx -180 ry 0 rz -11.91 deg; joints [26.427, -21.129, 63.851, -79.676, 100.405, 132.847]
  MoveL 1523 to (214.13, 422.55, -13.48) mm, rotated rx -180 ry 0 rz -11.91 deg; joints [26.433, -21.12, 63.831, -79.674, 100.412, 132.838]
  MoveL 1524 to (214.37, 422.59, -13.47) mm, rotated rx -180 ry 0 rz -11.91 deg; joints [26.439, -21.11, 63.81, -79.671, 100.418, 132.827]
  MoveL 1525 to (214.61, 422.65, -13.47) mm, rotated rx -180 ry 0 rz -11.91 deg; joints [26.445, -21.098, 63.785, -79.67, 100.425, 132.815]
  MoveL 1526 to (214.85, 422.74, -13.47) mm, rotated rx 180 ry 0 rz -11.91 deg; joints [26.451, -21.085, 63.758, -79.668, 100.431, 132.801]
  MoveL 1527 to (215.09, 422.84, -13.48) mm, rotated rx -180 ry 0 rz -11.91 deg; joints [26.456, -21.071, 63.728, -79.668, 100.438, 132.786]
  MoveL 1528 to (215.34, 422.97, -13.47) mm, rotated rx 180 ry 0 rz -11.91 deg; joints [26.461, -21.055, 63.694, -79.667, 100.445, 132.769]
  MoveL 1529 to (215.58, 423.13, -13.48) mm, rotated rx 180 ry 0 rz -11.91 deg; joints [26.465, -21.037, 63.656, -79.668, 100.452, 132.749]
  MoveL 1530 to (215.82, 423.33, -13.48) mm, rotated rx -180 ry 0 rz -11.91 deg; joints [26.469, -21.017, 63.614, -79.669, 100.458, 132.727]
  MoveL 1531 to (215.96, 423.46, -13.47) mm, rotated rx -180 ry 0 rz -11.91 deg; joints [26.471, -21.004, 63.586, -79.67, 100.463, 132.713]
  MoveL 1532 to (216.09, 423.6, -13.48) mm, rotated rx -180 ry 0 rz -11.91 deg; joints [26.473, -20.992, 63.559, -79.672, 100.466, 132.699]
  MoveL 1533 to (216.2, 423.73, -13.47) mm, rotated rx 180 ry 0 rz -11.91 deg; joints [26.474, -20.979, 63.533, -79.673, 100.47, 132.686]
  MoveL 1534 to (216.3, 423.87, -13.48) mm, rotated rx -180 ry 0 rz -11.91 deg; joints [26.475, -20.968, 63.508, -79.675, 100.473, 132.672]
  MoveL 1535 to (216.39, 424.01, -13.48) mm, rotated rx 180 ry 0 rz -11.91 deg; joints [26.476, -20.956, 63.483, -79.677, 100.476, 132.659]
  MoveL 1536 to (216.47, 424.15, -13.48) mm, rotated rx -180 ry 0 rz -11.91 deg; joints [26.476, -20.944, 63.459, -79.679, 100.478, 132.647]
  MoveL 1537 to (216.69, 424.27, -13.48) mm, rotated rx -180 ry 0 rz -11.91 deg; joints [26.48, -20.93, 63.428, -79.679, 100.484, 132.631]
  MoveL 1538 to (219.83, 424.27, -13.47) mm, rotated rx 180 ry 0 rz -11.91 deg; joints [26.567, -20.831, 63.216, -79.639, 100.568, 132.529]
  MoveL 1539 to (220.05, 424.15, -13.47) mm, rotated rx -180 ry 0 rz -11.91 deg; joints [26.575, -20.831, 63.217, -79.633, 100.573, 132.531]
  MoveL 1540 to (220.05, 53.41, -13.48) mm, rotated rx -180 ry 0 rz -11.91 deg; joints [32.836, -38.04, 100.626, -70.988, 99.147, 153.327]
  MoveL 1541 to (219.83, 53.17, -13.48) mm, rotated rx -180 ry 0 rz -11.91 deg; joints [32.833, -38.054, 100.657, -70.987, 99.141, 153.343]
  MoveL 1542 to (-197.29, 53.17, -13.47) mm, rotated rx -180 ry 0 rz -11.91 deg; joints [17.746, -44.608, 116.72, -84.232, 91.439, 161.337]
  MoveL 1543 to (-197.94, 53.17, -13.48) mm, rotated rx 180 ry 0 rz -11.91 deg; joints [17.719, -44.614, 116.737, -84.257, 91.43, 161.346]
  MoveL 1544 to (-198.16, 53.41, -13.48) mm, rotated rx 180 ry 0 rz -11.91 deg; joints [17.707, -44.609, 116.724, -84.268, 91.427, 161.338]
  MoveL 1545 to (-198.16, 424.15, -13.48) mm, rotated rx -180 ry 0 rz -11.91 deg; joints [13.889, -29.564, 82.255, -88.108, 90.94, 141.846]
  MoveL 1546 to (-198.01, 424.27, -13.47) mm, rotated rx -180 ry 0 rz -11.91 deg; joints [13.893, -29.556, 82.238, -88.105, 90.943, 141.836]
  MoveL 1547 to (-197.87, 424.15, -13.48) mm, rotated rx -180 ry 0 rz -11.91 deg; joints [13.899, -29.56, 82.247, -88.101, 90.946, 141.841]
  MoveL 1548 to (-197.73, 423.93, -13.47) mm, rotated rx -180 ry 0 rz -11.91 deg; joints [13.905, -29.57, 82.268, -88.095, 90.949, 141.853]
  MoveL 1549 to (-197.57, 423.71, -13.48) mm, rotated rx 180 ry 0 rz -11.91 deg; joints [13.912, -29.579, 82.288, -88.09, 90.953, 141.864]
  MoveL 1550 to (-197.38, 423.49, -13.47) mm, rotated rx -180 ry 0 rz -11.91 deg; joints [13.92, -29.588, 82.307, -88.083, 90.958, 141.874]
  MoveL 1551 to (-197.22, 423.33, -13.48) mm, rotated rx -180 ry 0 rz -11.91 deg; joints [13.926, -29.594, 82.32, -88.078, 90.961, 141.881]
  MoveL 1552 to (-197.14, 423.27, -13.48) mm, rotated rx -180 ry 0 rz -11.91 deg; joints [13.929, -29.596, 82.325, -88.075, 90.963, 141.884]
  MoveL 1553 to (-196.96, 423.13, -13.48) mm, rotated rx -180 ry 0 rz -11.91 deg; joints [13.936, -29.601, 82.336, -88.07, 90.967, 141.89]
  MoveL 1554 to (-196.78, 423, -13.48) mm, rotated rx -180 ry 0 rz -11.91 deg; joints [13.943, -29.605, 82.344, -88.064, 90.971, 141.894]
  MoveL 1555 to (-196.6, 422.9, -13.48) mm, rotated rx -180 ry 0 rz -11.91 deg; joints [13.95, -29.608, 82.351, -88.058, 90.975, 141.898]
  MoveL 1556 to (-196.42, 422.81, -13.48) mm, rotated rx -180 ry 0 rz -11.91 deg; joints [13.957, -29.611, 82.356, -88.053, 90.979, 141.901]
  MoveL 1557 to (-196.18, 422.71, -13.47) mm, rotated rx -180 ry 0 rz -11.91 deg; joints [13.966, -29.613, 82.36, -88.046, 90.984, 141.903]
  MoveL 1558 to (-195.93, 422.63, -13.47) mm, rotated rx -180 ry 0 rz -11.91 deg; joints [13.974, -29.614, 82.362, -88.039, 90.989, 141.904]
  MoveL 1559 to (-195.69, 422.58, -13.48) mm, rotated rx -180 ry 0 rz -11.91 deg; joints [13.982, -29.613, 82.361, -88.033, 90.995, 141.904]
  MoveL 1560 to (-195.45, 422.54, -13.48) mm, rotated rx -180 ry 0 rz -11.91 deg; joints [13.991, -29.612, 82.359, -88.026, 91, 141.903]
  MoveL 1561 to (-195.21, 422.52, -13.48) mm, rotated rx -180 ry 0 rz -11.91 deg; joints [13.999, -29.61, 82.354, -88.02, 91.004, 141.9]
  MoveL 1562 to (-194.97, 422.52, -13.48) mm, rotated rx 180 ry 0 rz -11.91 deg; joints [14.006, -29.607, 82.348, -88.014, 91.009, 141.897]
  Set speed (38.1 mm/s)
  MoveL 1563 to (-194.97, 421.25, -13.47) mm, rotated rx -180 ry 0 rz -11.91 deg; joints [14.017, -29.672, 82.489, -88.004, 91.013, 141.974]
  MoveL 1564 to (-195.61, 421.25, -13.47) mm, rotated rx -180 ry 0 rz -11.91 deg; joints [13.996, -29.68, 82.507, -88.02, 91, 141.983]
  Set speed (25.4 mm/s)
  MoveL 1565 to (-195.61, 421.25, -15.84) mm, rotated rx -180 ry 0 rz -11.91 deg; joints [13.997, -29.568, 82.481, -88.018, 90.998, 142.07]
  MoveL 1566 to (-195.61, 421.89, -16.48) mm, rotated rx -180 ry 0 rz -11.91 deg; joints [13.992, -29.506, 82.404, -88.023, 90.995, 142.054]
  Set speed (38.1 mm/s)
  MoveL 1567 to (-194.97, 422.52, -16.48) mm, rotated rx 180 ry 0 rz -11.91 deg; joints [14.007, -29.465, 82.315, -88.011, 91.006, 142.007]
  Set speed (76.2 mm/s)
  MoveL 1568 to (213.41, 422.52, -16.47) mm, rotated rx 180 ry 0 rz -11.91 deg; joints [26.414, -21.011, 63.846, -79.665, 100.376, 132.958]
  MoveL 1569 to (213.89, 422.53, -16.48) mm, rotated rx -180 ry 0 rz -11.91 deg; joints [26.428, -20.996, 63.813, -79.658, 100.389, 132.942]
  MoveL 1570 to (214.13, 422.55, -16.48) mm, rotated rx 180 ry 0 rz -11.91 deg; joints [26.434, -20.987, 63.794, -79.656, 100.395, 132.933]
  MoveL 1571 to (214.37, 422.59, -16.47) mm, rotated rx -180 ry 0 rz -11.91 deg; joints [26.44, -20.977, 63.772, -79.654, 100.402, 132.922]
  MoveL 1572 to (214.61, 422.65, -16.47) mm, rotated rx 180 ry 0 rz -11.91 deg; joints [26.446, -20.965, 63.747, -79.652, 100.408, 132.91]
  MoveL 1573 to (214.85, 422.74, -16.47) mm, rotated rx -180 ry 0 rz -11.91 deg; joints [26.452, -20.953, 63.72, -79.65, 100.415, 132.896]
  MoveL 1574 to (215.09, 422.84, -16.48) mm, rotated rx -180 ry 0 rz -11.91 deg; joints [26.457, -20.938, 63.69, -79.65, 100.422, 132.881]
  MoveL 1575 to (215.34, 422.97, -16.48) mm, rotated rx -180 ry 0 rz -11.91 deg; joints [26.462, -20.922, 63.656, -79.649, 100.428, 132.864]
  MoveL 1576 to (215.58, 423.13, -16.47) mm, rotated rx -180 ry 0 rz -11.91 deg; joints [26.466, -20.905, 63.618, -79.65, 100.435, 132.844]
  MoveL 1577 to (215.82, 423.33, -16.47) mm, rotated rx -180 ry 0 rz -11.91 deg; joints [26.47, -20.885, 63.576, -79.651, 100.442, 132.822]
  MoveL 1578 to (215.96, 423.46, -16.48) mm, rotated rx 180 ry 0 rz -11.91 deg; joints [26.472, -20.872, 63.548, -79.652, 100.446, 132.808]
  MoveL 1579 to (216.09, 423.6, -16.48) mm, rotated rx -180 ry 0 rz -11.91 deg; joints [26.474, -20.859, 63.521, -79.654, 100.45, 132.794]
  MoveL 1580 to (216.2, 423.73, -16.48) mm, rotated rx -180 ry 0 rz -11.91 deg; joints [26.475, -20.847, 63.495, -79.655, 100.453, 132.78]
  MoveL 1581 to (216.3, 423.87, -16.47) mm, rotated rx -180 ry 0 rz -11.91 deg; joints [26.476, -20.835, 63.47, -79.657, 100.456, 132.767]
  MoveL 1582 to (216.39, 424.01, -16.48) mm, rotated rx -180 ry 0 rz -11.91 deg; joints [26.477, -20.823, 63.445, -79.659, 100.459, 132.754]
  MoveL 1583 to (216.47, 424.15, -16.47) mm, rotated rx -180 ry 0 rz -11.91 deg; joints [26.477, -20.812, 63.421, -79.661, 100.462, 132.741]
  MoveL 1584 to (216.69, 424.27, -16.47) mm, rotated rx -180 ry 0 rz -11.91 deg; joints [26.481, -20.797, 63.39, -79.661, 100.468, 132.726]
  MoveL 1585 to (219.83, 424.27, -16.48) mm, rotated rx 180 ry 0 rz -11.91 deg; joints [26.568, -20.698, 63.178, -79.621, 100.551, 132.624]
  MoveL 1586 to (220.05, 424.15, -16.47) mm, rotated rx -180 ry 0 rz -11.91 deg; joints [26.576, -20.699, 63.179, -79.615, 100.557, 132.626]
  MoveL 1587 to (220.05, 53.41, -16.48) mm, rotated rx -180 ry 0 rz -11.91 deg; joints [32.837, -37.881, 100.596, -70.967, 99.106, 153.45]
  MoveL 1588 to (219.83, 53.17, -16.48) mm, rotated rx 180 ry 0 rz -11.91 deg; joints [32.835, -37.894, 100.626, -70.966, 99.099, 153.466]
  MoveL 1589 to (-196.42, 53.17, -16.47) mm, rotated rx -180 ry 0 rz -11.91 deg; joints [17.782, -44.414, 116.666, -84.194, 91.436, 161.477]
  MoveL 1590 to (-196.42, 53.41, -16.48) mm, rotated rx -180 ry 0 rz -11.91 deg; joints [17.779, -44.407, 116.647, -84.197, 91.436, 161.465]
  MoveL 1591 to (-196.42, 422.66, -16.48) mm, rotated rx 180 ry 0 rz -11.91 deg; joints [13.959, -29.476, 82.34, -88.05, 90.976, 142.02]
  MoveL 1592 to (-196.42, 422.81, -16.48) mm, rotated rx -180 ry 0 rz -11.91 deg; joints [13.958, -29.469, 82.324, -88.051, 90.976, 142.011]
  MoveL 1593 to (-196.18, 422.71, -16.48) mm, rotated rx 180 ry 0 rz -11.91 deg; joints [13.966, -29.471, 82.328, -88.044, 90.981, 142.013]
  MoveL 1594 to (-195.93, 422.63, -16.48) mm, rotated rx -180 ry 0 rz -11.91 deg; joints [13.975, -29.472, 82.33, -88.037, 90.986, 142.014]
  MoveL 1595 to (-195.69, 422.58, -16.48) mm, rotated rx -180 ry 0 rz -11.91 deg; joints [13.983, -29.472, 82.329, -88.03, 90.991, 142.014]
  MoveL 1596 to (-195.45, 422.54, -16.48) mm, rotated rx -180 ry 0 rz -11.91 deg; joints [13.991, -29.47, 82.327, -88.024, 90.996, 142.012]
  MoveL 1597 to (-195.21, 422.52, -16.48) mm, rotated rx 180 ry 0 rz -11.91 deg; joints [13.999, -29.468, 82.322, -88.017, 91.001, 142.01]
  MoveL 1598 to (-194.97, 422.52, -16.48) mm, rotated rx 180 ry 0 rz -11.91 deg; joints [14.007, -29.465, 82.315, -88.011, 91.006, 142.007]
  MoveL 1599 to (-164.9, 422.52, -17.53) mm, rotated rx -180 ry 0 rz -11.91 deg; joints [14.986, -29.026, 81.431, -87.243, 91.618, 141.587]
  MoveL 1600 to (213.41, 422.52, -17.53) mm, rotated rx -180 ry 0 rz -11.91 deg; joints [26.415, -20.965, 63.832, -79.658, 100.37, 132.991]
  MoveL 1601 to (213.89, 422.53, -17.53) mm, rotated rx -180 ry 0 rz -11.91 deg; joints [26.428, -20.949, 63.799, -79.652, 100.383, 132.975]
  MoveL 1602 to (214.13, 422.55, -17.53) mm, rotated rx -180 ry 0 rz -11.91 deg; joints [26.434, -20.94, 63.78, -79.65, 100.39, 132.966]
  MoveL 1603 to (214.37, 422.59, -17.53) mm, rotated rx -180 ry 0 rz -11.91 deg; joints [26.441, -20.93, 63.758, -79.647, 100.396, 132.955]
  MoveL 1604 to (214.61, 422.65, -17.52) mm, rotated rx 180 ry 0 rz -11.91 deg; joints [26.446, -20.919, 63.734, -79.646, 100.403, 132.943]
  MoveL 1605 to (214.85, 422.74, -17.53) mm, rotated rx 180 ry 0 rz -11.91 deg; joints [26.452, -20.906, 63.707, -79.644, 100.409, 132.929]
  MoveL 1606 to (215.09, 422.84, -17.53) mm, rotated rx 180 ry 0 rz -11.91 deg; joints [26.457, -20.892, 63.676, -79.643, 100.416, 132.914]
  MoveL 1607 to (215.34, 422.97, -17.53) mm, rotated rx 180 ry 0 rz -11.91 deg; joints [26.462, -20.876, 63.642, -79.643, 100.423, 132.897]
  MoveL 1608 to (215.58, 423.13, -17.53) mm, rotated rx -180 ry 0 rz -11.91 deg; joints [26.467, -20.858, 63.605, -79.644, 100.43, 132.877]
  MoveL 1609 to (215.82, 423.33, -17.52) mm, rotated rx -180 ry 0 rz -11.91 deg; joints [26.471, -20.838, 63.562, -79.645, 100.436, 132.855]
  MoveL 1610 to (215.96, 423.46, -17.53) mm, rotated rx 180 ry 0 rz -11.91 deg; joints [26.473, -20.825, 63.535, -79.646, 100.441, 132.841]
  MoveL 1611 to (216.09, 423.6, -17.53) mm, rotated rx -180 ry 0 rz -11.91 deg; joints [26.474, -20.812, 63.508, -79.648, 100.444, 132.827]
  MoveL 1612 to (216.2, 423.73, -17.53) mm, rotated rx -180 ry 0 rz -11.91 deg; joints [26.475, -20.8, 63.482, -79.649, 100.448, 132.814]
  MoveL 1613 to (216.3, 423.87, -17.52) mm, rotated rx 180 ry 0 rz -11.91 deg; joints [26.476, -20.788, 63.457, -79.651, 100.451, 132.8]
  MoveL 1614 to (216.39, 424.01, -17.52) mm, rotated rx 180 ry 0 rz -11.91 deg; joints [26.477, -20.777, 63.432, -79.653, 100.454, 132.787]
  MoveL 1615 to (216.47, 424.15, -17.53) mm, rotated rx -180 ry 0 rz -11.91 deg; joints [26.477, -20.765, 63.408, -79.655, 100.456, 132.775]
  MoveL 1616 to (216.69, 424.27, -17.53) mm, rotated rx -180 ry 0 rz -11.91 deg; joints [26.482, -20.751, 63.377, -79.655, 100.462, 132.759]
  MoveL 1617 to (219.83, 424.27, -17.52) mm, rotated rx -180 ry 0 rz -11.91 deg; joints [26.569, -20.652, 63.164, -79.615, 100.546, 132.657]
  MoveL 1618 to (220.05, 424.15, -17.52) mm, rotated rx -180 ry 0 rz -11.91 deg; joints [26.577, -20.652, 63.165, -79.609, 100.551, 132.659]
  MoveL 1619 to (220.05, 53.41, -17.52) mm, rotated rx -180 ry 0 rz -11.91 deg; joints [32.838, -37.825, 100.585, -70.96, 99.091, 153.493]
  MoveL 1620 to (219.83, 53.17, -17.53) mm, rotated rx -180 ry 0 rz -11.91 deg; joints [32.835, -37.838, 100.616, -70.959, 99.085, 153.51]
  MoveL 1621 to (-195.15, 53.17, -17.53) mm, rotated rx 180 ry 0 rz -11.91 deg; joints [17.834, -44.337, 116.621, -84.143, 91.448, 161.511]
  MoveL 1622 to (-195.65, 53.17, -17.52) mm, rotated rx -180 ry 0 rz -11.91 deg; joints [17.814, -44.342, 116.634, -84.162, 91.442, 161.518]
  MoveL 1623 to (-195.81, 53.41, -17.53) mm, rotated rx 180 ry 0 rz -11.91 deg; joints [17.804, -44.336, 116.62, -84.172, 91.439, 161.51]
  MoveL 1624 to (-195.81, 422.38, -17.52) mm, rotated rx -180 ry 0 rz -11.91 deg; joints [13.981, -29.434, 82.343, -88.031, 90.988, 142.066]
  MoveL 1625 to (-195.65, 422.57, -17.53) mm, rotated rx -180 ry 0 rz -11.91 deg; joints [13.985, -29.422, 82.317, -88.028, 90.991, 142.052]
  MoveL 1626 to (-195.48, 422.55, -17.53) mm, rotated rx 180 ry 0 rz -11.91 deg; joints [13.991, -29.421, 82.316, -88.024, 90.994, 142.051]
  MoveL 1627 to (-195.32, 422.53, -17.52) mm, rotated rx -180 ry 0 rz -11.91 deg; joints [13.996, -29.42, 82.313, -88.019, 90.998, 142.049]
  MoveL 1628 to (-195.15, 422.52, -17.53) mm, rotated rx -180 ry 0 rz -11.91 deg; joints [14.002, -29.418, 82.309, -88.015, 91.001, 142.047]
  MoveL 1629 to (-194.97, 422.52, -17.52) mm, rotated rx -180 ry 0 rz -11.91 deg; joints [14.007, -29.416, 82.304, -88.01, 91.005, 142.045]
  MoveL 1630 to (-164.9, 422.52, -17.53) mm, rotated rx -180 ry 0 rz -11.91 deg; joints [14.986, -29.026, 81.431, -87.243, 91.618, 141.587]
  Set speed (38.1 mm/s)
  MoveL 1631 to (-164.28, 421.77, -17.52) mm, rotated rx -180 ry 0 rz -11.91 deg; joints [15.012, -29.056, 81.496, -87.221, 91.632, 141.623]
  MoveL 1632 to (-164.81, 418.84, -17.52) mm, rotated rx -180 ry 0 rz -11.91 deg; joints [15.021, -29.214, 81.841, -87.209, 91.628, 141.81]
  MoveL 1633 to (-164.93, 418.21, -16.89) mm, rotated rx -180 ry 0 rz -11.91 deg; joints [15.022, -29.277, 81.921, -87.207, 91.628, 141.826]
  Set speed (100.0 mm/s)
  MoveL 1634 to (-164.93, 418.21, 24.52) mm, rotated rx 180 ry 0 rz -11.91 deg; joints [15.011, -31.202, 82.299, -87.261, 91.696, 140.281]
  MoveL 1635 to (-164.87, 434.05, 24.52) mm, rotated rx 180 ry 0 rz -11.91 deg; joints [14.876, -30.363, 80.516, -87.393, 91.655, 139.332]
  MoveL 1636 to (-164.87, 434.05, -6.52) mm, rotated rx -180 ry 0 rz -11.91 deg; joints [14.884, -28.94, 80.243, -87.354, 91.607, 140.483]
  Set speed (25.4 mm/s)
  MoveL 1637 to (-164.87, 434.05, -9.84) mm, rotated rx -180 ry 0 rz -11.91 deg; joints [14.885, -28.785, 80.209, -87.35, 91.602, 140.603]
  MoveL 1638 to (-164.72, 433.43, -10.48) mm, rotated rx -180 ry 0 rz -11.91 deg; joints [14.895, -28.786, 80.269, -87.341, 91.606, 140.662]
  Set speed (38.1 mm/s)
  MoveL 1639 to (-164.28, 431.48, -10.47) mm, rotated rx 180 ry 0 rz -11.91 deg; joints [14.926, -28.882, 80.477, -87.313, 91.62, 140.775]
  MoveL 1640 to (-164.9, 430.7, -10.48) mm, rotated rx -180 ry 0 rz -11.91 deg; joints [14.913, -28.931, 80.584, -87.322, 91.609, 140.832]
  Set speed (76.2 mm/s)
  MoveL 1641 to (-194.97, 430.7, -10.47) mm, rotated rx -180 ry 0 rz -11.91 deg; joints [13.939, -29.327, 81.462, -88.078, 90.989, 141.291]
  MoveL 1642 to (-202.2, 430.7, -10.48) mm, rotated rx 180 ry 0 rz -11.91 deg; joints [13.703, -29.417, 81.663, -88.262, 90.841, 141.397]
  MoveL 1643 to (-203.17, 430.7, -10.47) mm, rotated rx -180 ry 0 rz -11.91 deg; joints [13.672, -29.429, 81.69, -88.287, 90.821, 141.411]
  MoveL 1644 to (-203.41, 430.69, -10.48) mm, rotated rx 180 ry 0 rz -11.91 deg; joints [13.664, -29.433, 81.698, -88.293, 90.816, 141.416]
  MoveL 1645 to (-203.65, 430.65, -10.48) mm, rotated rx 180 ry 0 rz -11.91 deg; joints [13.657, -29.437, 81.709, -88.299, 90.812, 141.421]
  MoveL 1646 to (-203.89, 430.6, -10.48) mm, rotated rx 180 ry 0 rz -11.91 deg; joints [13.649, -29.443, 81.722, -88.305, 90.807, 141.428]
  MoveL 1647 to (-204.13, 430.52, -10.48) mm, rotated rx -180 ry 0 rz -11.91 deg; joints [13.642, -29.45, 81.736, -88.31, 90.802, 141.436]
  MoveL 1648 to (-204.42, 430.43, -10.47) mm, rotated rx 180 ry 0 rz -11.91 deg; joints [13.633, -29.459, 81.755, -88.317, 90.797, 141.446]
  MoveL 1649 to (-204.57, 430.37, -10.48) mm, rotated rx -180 ry 0 rz -11.91 deg; joints [13.629, -29.463, 81.765, -88.32, 90.794, 141.452]
  MoveL 1650 to (-204.72, 430.31, -10.48) mm, rotated rx -180 ry 0 rz -11.91 deg; joints [13.625, -29.468, 81.777, -88.324, 90.791, 141.458]
  MoveL 1651 to (-204.86, 430.23, -10.48) mm, rotated rx 180 ry 0 rz -11.91 deg; joints [13.62, -29.474, 81.789, -88.327, 90.788, 141.464]
  MoveL 1652 to (-205.01, 430.15, -10.47) mm, rotated rx 180 ry 0 rz -11.91 deg; joints [13.616, -29.48, 81.803, -88.33, 90.785, 141.472]
  MoveL 1653 to (-205.16, 430.05, -10.48) mm, rotated rx 180 ry 0 rz -11.91 deg; joints [13.612, -29.487, 81.817, -88.333, 90.783, 141.48]
  MoveL 1654 to (-205.3, 429.94, -10.48) mm, rotated rx 180 ry 0 rz -11.91 deg; joints [13.608, -29.494, 81.834, -88.336, 90.78, 141.488]
  MoveL 1655 to (-205.53, 429.75, -10.48) mm, rotated rx -180 ry 0 rz -11.91 deg; joints [13.603, -29.507, 81.861, -88.34, 90.776, 141.503]
  MoveL 1656 to (-205.75, 429.52, -10.47) mm, rotated rx -180 ry 0 rz -11.91 deg; joints [13.597, -29.522, 81.894, -88.345, 90.772, 141.521]
  MoveL 1657 to (-205.92, 429.3, -10.47) mm, rotated rx -180 ry 0 rz -11.91 deg; joints [13.593, -29.535, 81.922, -88.347, 90.77, 141.536]
  MoveL 1658 to (-206.06, 429.09, -10.48) mm, rotated rx -180 ry 0 rz -11.91 deg; joints [13.59, -29.548, 81.95, -88.349, 90.767, 141.551]
  MoveL 1659 to (-206.14, 428.95, -10.47) mm, rotated rx 180 ry 0 rz -11.91 deg; joints [13.589, -29.556, 81.967, -88.35, 90.766, 141.56]
  MoveL 1660 to (-206.21, 428.82, -10.47) mm, rotated rx 180 ry 0 rz -11.91 deg; joints [13.588, -29.564, 81.984, -88.351, 90.765, 141.57]
  MoveL 1661 to (-206.27, 428.69, -10.48) mm, rotated rx -180 ry 0 rz -11.91 deg; joints [13.587, -29.571, 82.001, -88.352, 90.764, 141.579]
  MoveL 1662 to (-206.32, 428.55, -10.47) mm, rotated rx -180 ry 0 rz -11.91 deg; joints [13.586, -29.579, 82.018, -88.352, 90.764, 141.588]
  MoveL 1663 to (-206.37, 428.42, -10.47) mm, rotated rx 180 ry 0 rz -11.91 deg; joints [13.586, -29.586, 82.034, -88.353, 90.763, 141.597]
  MoveL 1664 to (-206.41, 428.28, -10.48) mm, rotated rx -180 ry 0 rz -11.91 deg; joints [13.585, -29.594, 82.05, -88.353, 90.763, 141.605]
  MoveL 1665 to (-206.47, 428.01, -10.47) mm, rotated rx -180 ry 0 rz -11.91 deg; joints [13.586, -29.609, 82.082, -88.352, 90.762, 141.623]
  MoveL 1666 to (-206.5, 427.77, -10.48) mm, rotated rx -180 ry 0 rz -11.91 deg; joints [13.586, -29.621, 82.11, -88.351, 90.762, 141.638]
  MoveL 1667 to (-206.52, 427.53, -10.47) mm, rotated rx -180 ry 0 rz -11.91 deg; joints [13.588, -29.634, 82.138, -88.35, 90.763, 141.653]
  MoveL 1668 to (-206.52, 427.04, -10.47) mm, rotated rx -180 ry 0 rz -11.91 deg; joints [13.592, -29.659, 82.192, -88.347, 90.764, 141.682]
  MoveL 1669 to (-206.52, 50.21, -10.48) mm, rotated rx -180 ry 0 rz -11.91 deg; joints [17.407, -44.98, 117.224, -84.551, 91.323, 161.458]
  MoveL 1670 to (-206.51, 49.73, -10.47) mm, rotated rx -180 ry 0 rz -11.91 deg; joints [17.414, -44.995, 117.262, -84.544, 91.323, 161.481]
  MoveL 1671 to (-206.48, 49.48, -10.48) mm, rotated rx -180 ry 0 rz -11.91 deg; joints [17.418, -45.003, 117.281, -84.539, 91.323, 161.492]
  MoveL 1672 to (-206.43, 49.24, -10.48) mm, rotated rx -180 ry 0 rz -11.91 deg; joints [17.424, -45.01, 117.299, -84.534, 91.324, 161.503]
  MoveL 1673 to (-206.37, 49.02, -10.47) mm, rotated rx -180 ry 0 rz -11.91 deg; joints [17.429, -45.017, 117.315, -84.529, 91.325, 161.513]
  MoveL 1674 to (-206.28, 48.8, -10.47) mm, rotated rx -180 ry 0 rz -11.91 deg; joints [17.435, -45.023, 117.331, -84.523, 91.326, 161.523]
  MoveL 1675 to (-206.18, 48.57, -10.47) mm, rotated rx -180 ry 0 rz -11.91 deg; joints [17.442, -45.029, 117.346, -84.516, 91.327, 161.532]
  MoveL 1676 to (-206.06, 48.35, -10.48) mm, rotated rx -180 ry 0 rz -11.91 deg; joints [17.45, -45.035, 117.361, -84.508, 91.328, 161.541]
  MoveL 1677 to (-205.98, 48.22, -10.48) mm, rotated rx -180 ry 0 rz -11.91 deg; joints [17.455, -45.039, 117.369, -84.503, 91.329, 161.546]
  MoveL 1678 to (-205.88, 48.09, -10.48) mm, rotated rx -180 ry 0 rz -11.91 deg; joints [17.461, -45.042, 117.377, -84.498, 91.331, 161.551]
  MoveL 1679 to (-205.78, 47.96, -10.48) mm, rotated rx 180 ry 0 rz -11.91 deg; joints [17.467, -45.045, 117.385, -84.492, 91.332, 161.555]
  MoveL 1680 to (-205.66, 47.83, -10.48) mm, rotated rx -180 ry 0 rz -11.91 deg; joints [17.473, -45.048, 117.393, -84.486, 91.333, 161.56]
  MoveL 1681 to (-205.51, 47.67, -10.48) mm, rotated rx -180 ry 0 rz -11.91 deg; joints [17.482, -45.052, 117.401, -84.478, 91.336, 161.565]
  MoveL 1682 to (-205.35, 47.54, -10.47) mm, rotated rx -180 ry 0 rz -11.91 deg; joints [17.49, -45.055, 117.408, -84.47, 91.338, 161.57]
  MoveL 1683 to (-205.19, 47.42, -10.47) mm, rotated rx 180 ry 0 rz -11.91 deg; joints [17.498, -45.057, 117.414, -84.462, 91.34, 161.573]
  MoveL 1684 to (-205.03, 47.31, -10.47) mm, rotated rx -180 ry 0 rz -11.91 deg; joints [17.506, -45.059, 117.418, -84.455, 91.342, 161.576]
  MoveL 1685 to (-204.81, 47.18, -10.47) mm, rotated rx -180 ry 0 rz -11.91 deg; joints [17.516, -45.061, 117.423, -84.444, 91.345, 161.579]
  MoveL 1686 to (-204.58, 47.08, -10.47) mm, rotated rx 180 ry 0 rz -11.91 deg; joints [17.527, -45.062, 117.426, -84.434, 91.348, 161.581]
  MoveL 1687 to (-204.36, 46.99, -10.48) mm, rotated rx 180 ry 0 rz -11.91 deg; joints [17.537, -45.063, 117.427, -84.424, 91.351, 161.582]
  MoveL 1688 to (-204.13, 46.92, -10.48) mm, rotated rx -180 ry 0 rz -11.91 deg; joints [17.547, -45.063, 117.427, -84.415, 91.354, 161.581]
  MoveL 1689 to (-203.89, 46.87, -10.47) mm, rotated rx -180 ry 0 rz -11.91 deg; joints [17.558, -45.062, 117.425, -84.405, 91.357, 161.58]
  MoveL 1690 to (-203.65, 46.84, -10.48) mm, rotated rx -180 ry 0 rz -11.91 deg; joints [17.568, -45.061, 117.421, -84.395, 91.361, 161.579]
  MoveL 1691 to (-203.41, 46.83, -10.48) mm, rotated rx -180 ry 0 rz -11.91 deg; joints [17.578, -45.059, 117.416, -84.385, 91.364, 161.576]
  MoveL 1692 to (-203.17, 46.82, -10.47) mm, rotated rx 180 ry 0 rz -11.91 deg; joints [17.588, -45.057, 117.41, -84.376, 91.367, 161.572]
  MoveL 1693 to (222.09, 46.82, -10.48) mm, rotated rx 180 ry 0 rz -11.91 deg; joints [33.033, -38.386, 101.076, -70.791, 99.199, 153.456]
  MoveL 1694 to (223.29, 46.83, -10.48) mm, rotated rx -180 ry 0 rz -11.91 deg; joints [33.071, -38.36, 101.014, -70.762, 99.227, 153.428]
  MoveL 1695 to (223.53, 46.84, -10.47) mm, rotated rx -180 ry 0 rz -11.91 deg; joints [33.079, -38.354, 101, -70.757, 99.233, 153.422]
  MoveL 1696 to (223.77, 46.87, -10.47) mm, rotated rx -180 ry 0 rz -11.91 deg; joints [33.086, -38.347, 100.985, -70.752, 99.239, 153.414]
  MoveL 1697 to (224.01, 46.92, -10.48) mm, rotated rx -180 ry 0 rz -11.91 deg; joints [33.092, -38.34, 100.969, -70.747, 99.245, 153.406]
  MoveL 1698 to (224.24, 46.99, -10.48) mm, rotated rx -180 ry 0 rz -11.91 deg; joints [33.098, -38.333, 100.952, -70.744, 99.251, 153.398]
  MoveL 1699 to (224.46, 47.08, -10.48) mm, rotated rx -180 ry 0 rz -11.91 deg; joints [33.103, -38.325, 100.933, -70.74, 99.256, 153.389]
  MoveL 1700 to (224.69, 47.18, -10.48) mm, rotated rx 180 ry 0 rz -11.91 deg; joints [33.108, -38.316, 100.913, -70.738, 99.262, 153.379]
  MoveL 1701 to (224.92, 47.31, -10.48) mm, rotated rx -180 ry 0 rz -11.91 deg; joints [33.112, -38.306, 100.891, -70.735, 99.268, 153.368]
  MoveL 1702 to (225.07, 47.42, -10.48) mm, rotated rx 180 ry 0 rz -11.91 deg; joints [33.115, -38.299, 100.874, -70.734, 99.273, 153.359]
  MoveL 1703 to (225.23, 47.54, -10.48) mm, rotated rx -180 ry 0 rz -11.91 deg; joints [33.118, -38.291, 100.857, -70.734, 99.277, 153.35]
  MoveL 1704 to (225.39, 47.67, -10.47) mm, rotated rx -180 ry 0 rz -11.91 deg; joints [33.12, -38.283, 100.837, -70.733, 99.281, 153.34]
  MoveL 1705 to (225.55, 47.83, -10.48) mm, rotated rx 180 ry 0 rz -11.91 deg; joints [33.122, -38.274, 100.817, -70.734, 99.286, 153.329]
  MoveL 1706 to (225.66, 47.96, -10.47) mm, rotated rx -180 ry 0 rz -11.91 deg; joints [33.123, -38.267, 100.8, -70.734, 99.29, 153.32]
  MoveL 1707 to (225.77, 48.09, -10.48) mm, rotated rx 180 ry 0 rz -11.91 deg; joints [33.123, -38.26, 100.785, -70.735, 99.293, 153.312]
  MoveL 1708 to (225.86, 48.22, -10.48) mm, rotated rx 180 ry 0 rz -11.91 deg; joints [33.123, -38.253, 100.769, -70.736, 99.296, 153.304]
  MoveL 1709 to (225.94, 48.35, -10.48) mm, rotated rx 180 ry 0 rz -11.91 deg; joints [33.123, -38.247, 100.755, -70.737, 99.298, 153.296]
  MoveL 1710 to (226.07, 48.57, -10.48) mm, rotated rx 180 ry 0 rz -11.91 deg; joints [33.123, -38.236, 100.73, -70.74, 99.303, 153.283]
  MoveL 1711 to (226.17, 48.8, -10.47) mm, rotated rx -180 ry 0 rz -11.91 deg; joints [33.121, -38.226, 100.707, -70.743, 99.306, 153.27]
  MoveL 1712 to (226.25, 49.02, -10.48) mm, rotated rx 180 ry 0 rz -11.91 deg; joints [33.119, -38.217, 100.685, -70.747, 99.309, 153.258]
  MoveL 1713 to (226.31, 49.24, -10.48) mm, rotated rx 180 ry 0 rz -11.91 deg; joints [33.117, -38.207, 100.664, -70.751, 99.312, 153.246]
  MoveL 1714 to (226.36, 49.48, -10.48) mm, rotated rx -180 ry 0 rz -11.91 deg; joints [33.113, -38.198, 100.642, -70.756, 99.315, 153.234]
  MoveL 1715 to (226.39, 49.73, -10.47) mm, rotated rx 180 ry 0 rz -11.91 deg; joints [33.109, -38.188, 100.622, -70.762, 99.317, 153.222]
  MoveL 1716 to (226.4, 50.21, -10.47) mm, rotated rx -180 ry 0 rz -11.91 deg; joints [33.1, -38.171, 100.582, -70.774, 99.32, 153.2]
  MoveL 1717 to (226.4, 427.53, -10.48) mm, rotated rx -180 ry 0 rz -11.91 deg; joints [26.703, -20.54, 62.357, -79.65, 100.769, 131.979]
  MoveL 1718 to (226.39, 427.77, -10.48) mm, rotated rx -180 ry 0 rz -11.91 deg; joints [26.699, -20.525, 62.324, -79.656, 100.769, 131.961]
  MoveL 1719 to (226.37, 428.01, -10.48) mm, rotated rx -180 ry 0 rz -11.91 deg; joints [26.695, -20.51, 62.293, -79.662, 100.769, 131.944]
  MoveL 1720 to (226.34, 428.16, -10.47) mm, rotated rx -180 ry 0 rz -11.91 deg; joints [26.692, -20.501, 62.275, -79.665, 100.769, 131.934]
  MoveL 1721 to (226.31, 428.3, -10.48) mm, rotated rx -180 ry 0 rz -11.91 deg; joints [26.689, -20.493, 62.257, -79.669, 100.768, 131.924]
  MoveL 1722 to (226.27, 428.45, -10.48) mm, rotated rx -180 ry 0 rz -11.91 deg; joints [26.686, -20.484, 62.24, -79.673, 100.768, 131.915]
  MoveL 1723 to (226.22, 428.59, -10.48) mm, rotated rx -180 ry 0 rz -11.91 deg; joints [26.683, -20.476, 62.223, -79.677, 100.767, 131.906]
  MoveL 1724 to (226.16, 428.74, -10.47) mm, rotated rx -180 ry 0 rz -11.91 deg; joints [26.679, -20.469, 62.207, -79.681, 100.766, 131.897]
  MoveL 1725 to (226.1, 428.89, -10.48) mm, rotated rx 180 ry 0 rz -11.91 deg; joints [26.676, -20.461, 62.191, -79.685, 100.764, 131.888]
  MoveL 1726 to (226.03, 429.03, -10.47) mm, rotated rx 180 ry 0 rz -11.91 deg; joints [26.671, -20.454, 62.176, -79.689, 100.763, 131.88]
  MoveL 1727 to (225.94, 429.18, -10.47) mm, rotated rx 180 ry 0 rz -11.91 deg; joints [26.667, -20.447, 62.162, -79.694, 100.761, 131.872]
  MoveL 1728 to (225.82, 429.37, -10.48) mm, rotated rx 180 ry 0 rz -11.91 deg; joints [26.661, -20.439, 62.144, -79.7, 100.758, 131.861]
  MoveL 1729 to (225.67, 429.56, -10.48) mm, rotated rx -180 ry 0 rz -11.91 deg; joints [26.654, -20.431, 62.128, -79.706, 100.755, 131.852]
  MoveL 1730 to (225.5, 429.75, -10.48) mm, rotated rx 180 ry 0 rz -11.91 deg; joints [26.647, -20.424, 62.114, -79.713, 100.75, 131.844]
  MoveL 1731 to (225.29, 429.94, -10.48) mm, rotated rx -180 ry 0 rz -11.91 deg; joints [26.639, -20.418, 62.101, -79.719, 100.745, 131.836]
  MoveL 1732 to (225.13, 430.07, -10.48) mm, rotated rx -180 ry 0 rz -11.91 deg; joints [26.632, -20.415, 62.095, -79.724, 100.741, 131.832]
  MoveL 1733 to (224.97, 430.18, -10.48) mm, rotated rx -180 ry 0 rz -11.91 deg; joints [26.626, -20.413, 62.09, -79.729, 100.737, 131.829]
  MoveL 1734 to (224.81, 430.28, -10.48) mm, rotated rx 180 ry 0 rz -11.91 deg; joints [26.621, -20.412, 62.088, -79.733, 100.733, 131.827]
  MoveL 1735 to (224.65, 430.37, -10.48) mm, rotated rx -180 ry 0 rz -11.91 deg; joints [26.615, -20.411, 62.087, -79.737, 100.729, 131.826]
  MoveL 1736 to (224.49, 430.44, -10.48) mm, rotated rx -180 ry 0 rz -11.91 deg; joints [26.61, -20.411, 62.088, -79.741, 100.725, 131.825]
  MoveL 1737 to (224.33, 430.51, -10.48) mm, rotated rx 180 ry 0 rz -11.91 deg; joints [26.604, -20.412, 62.09, -79.744, 100.721, 131.826]
  MoveL 1738 to (224.17, 430.56, -10.48) mm, rotated rx -180 ry 0 rz -11.91 deg; joints [26.599, -20.414, 62.094, -79.747, 100.717, 131.827]
  MoveL 1739 to (224.01, 430.6, -10.48) mm, rotated rx -180 ry 0 rz -11.91 deg; joints [26.594, -20.416, 62.098, -79.75, 100.713, 131.829]
  MoveL 1740 to (223.77, 430.66, -10.47) mm, rotated rx 180 ry 0 rz -11.91 deg; joints [26.587, -20.421, 62.108, -79.754, 100.707, 131.833]
  MoveL 1741 to (223.53, 430.69, -10.47) mm, rotated rx -180 ry 0 rz -11.91 deg; joints [26.58, -20.426, 62.12, -79.758, 100.7, 131.839]
  MoveL 1742 to (223.29, 430.7, -10.47) mm, rotated rx 180 ry 0 rz -11.91 deg; joints [26.573, -20.433, 62.135, -79.761, 100.694, 131.846]
  MoveL 1743 to (223.05, 430.7, -10.47) mm, rotated rx -180 ry 0 rz -11.91 deg; joints [26.566, -20.441, 62.152, -79.764, 100.687, 131.854]
  MoveL 1744 to (-164.9, 430.7, -10.48) mm, rotated rx -180 ry 0 rz -11.91 deg; joints [14.913, -28.931, 80.584, -87.322, 91.609, 140.832]
  Set speed (38.1 mm/s)
  MoveL 1745 to (-165.25, 431.87, -10.48) mm, rotated rx -180 ry 0 rz -11.91 deg; joints [14.891, -28.875, 80.462, -87.341, 91.598, 140.766]
  MoveL 1746 to (-164.27, 432.52, -10.48) mm, rotated rx -180 ry 0 rz -11.91 deg; joints [14.917, -28.827, 80.357, -87.322, 91.617, 140.71]
  Set speed (25.4 mm/s)
  MoveL 1747 to (-164.27, 432.52, -12.84) mm, rotated rx -180 ry 0 rz -11.91 deg; joints [14.918, -28.717, 80.332, -87.319, 91.614, 140.796]
  MoveL 1748 to (-164.27, 431.89, -13.47) mm, rotated rx 180 ry 0 rz -11.91 deg; joints [14.924, -28.721, 80.398, -87.313, 91.614, 140.858]
  Set speed (38.1 mm/s)
  MoveL 1749 to (-164.9, 431.25, -13.48) mm, rotated rx -180 ry 0 rz -11.91 deg; joints [14.909, -28.763, 80.489, -87.323, 91.603, 140.907]
  Set speed (76.2 mm/s)
  MoveL 1750 to (-194.97, 431.25, -13.48) mm, rotated rx -180 ry 0 rz -11.91 deg; joints [13.935, -29.157, 81.368, -88.079, 90.984, 141.366]
  MoveL 1751 to (-201.24, 431.25, -13.48) mm, rotated rx 180 ry 0 rz -11.91 deg; joints [13.731, -29.236, 81.543, -88.239, 90.856, 141.459]
  MoveL 1752 to (-201.48, 431.25, -13.47) mm, rotated rx -180 ry 0 rz -11.91 deg; joints [13.723, -29.239, 81.55, -88.245, 90.851, 141.463]
  MoveL 1753 to (-201.72, 431.23, -13.47) mm, rotated rx -180 ry 0 rz -11.91 deg; joints [13.716, -29.243, 81.559, -88.251, 90.846, 141.467]
  MoveL 1754 to (-201.96, 431.19, -13.48) mm, rotated rx -180 ry 0 rz -11.91 deg; joints [13.708, -29.248, 81.57, -88.257, 90.842, 141.473]
  MoveL 1755 to (-202.2, 431.13, -13.48) mm, rotated rx 180 ry 0 rz -11.91 deg; joints [13.701, -29.254, 81.583, -88.263, 90.837, 141.48]
  MoveL 1756 to (-204.13, 430.52, -13.48) mm, rotated rx 180 ry 0 rz -11.91 deg; joints [13.643, -29.309, 81.705, -88.308, 90.799, 141.546]
  MoveL 1757 to (-204.42, 430.43, -13.48) mm, rotated rx 180 ry 0 rz -11.91 deg; joints [13.634, -29.318, 81.724, -88.315, 90.794, 141.556]
  MoveL 1758 to (-204.57, 430.37, -13.48) mm, rotated rx -180 ry 0 rz -11.91 deg; joints [13.63, -29.322, 81.734, -88.318, 90.791, 141.561]
  MoveL 1759 to (-204.72, 430.31, -13.47) mm, rotated rx -180 ry 0 rz -11.91 deg; joints [13.625, -29.327, 81.745, -88.322, 90.788, 141.567]
  MoveL 1760 to (-204.86, 430.23, -13.48) mm, rotated rx -180 ry 0 rz -11.91 deg; joints [13.621, -29.333, 81.758, -88.325, 90.785, 141.574]
  MoveL 1761 to (-205.01, 430.15, -13.48) mm, rotated rx -180 ry 0 rz -11.91 deg; joints [13.617, -29.339, 81.771, -88.328, 90.783, 141.581]
  MoveL 1762 to (-205.16, 430.05, -13.48) mm, rotated rx -180 ry 0 rz -11.91 deg; joints [13.613, -29.346, 81.786, -88.331, 90.78, 141.589]
  MoveL 1763 to (-205.3, 429.94, -13.48) mm, rotated rx -180 ry 0 rz -11.91 deg; joints [13.609, -29.353, 81.802, -88.334, 90.777, 141.598]
  MoveL 1764 to (-205.53, 429.75, -13.48) mm, rotated rx 180 ry 0 rz -11.91 deg; joints [13.603, -29.366, 81.83, -88.338, 90.773, 141.613]
  MoveL 1765 to (-205.75, 429.52, -13.48) mm, rotated rx 180 ry 0 rz -11.91 deg; joints [13.598, -29.381, 81.862, -88.342, 90.77, 141.63]
  MoveL 1766 to (-205.92, 429.3, -13.48) mm, rotated rx -180 ry 0 rz -11.91 deg; joints [13.594, -29.394, 81.891, -88.345, 90.767, 141.646]
  MoveL 1767 to (-206.06, 429.09, -13.48) mm, rotated rx -180 ry 0 rz -11.91 deg; joints [13.591, -29.407, 81.919, -88.347, 90.765, 141.661]
  MoveL 1768 to (-206.14, 428.95, -13.48) mm, rotated rx -180 ry 0 rz -11.91 deg; joints [13.59, -29.415, 81.936, -88.348, 90.764, 141.67]
  MoveL 1769 to (-206.21, 428.82, -13.48) mm, rotated rx 180 ry 0 rz -11.91 deg; joints [13.589, -29.422, 81.953, -88.349, 90.763, 141.679]
  MoveL 1770 to (-206.27, 428.69, -13.48) mm, rotated rx -180 ry 0 rz -11.91 deg; joints [13.588, -29.43, 81.97, -88.35, 90.762, 141.688]
  MoveL 1771 to (-206.32, 428.55, -13.47) mm, rotated rx -180 ry 0 rz -11.91 deg; joints [13.587, -29.438, 81.986, -88.35, 90.761, 141.697]
  MoveL 1772 to (-206.37, 428.42, -13.47) mm, rotated rx -180 ry 0 rz -11.91 deg; joints [13.586, -29.445, 82.003, -88.351, 90.76, 141.706]
  MoveL 1773 to (-206.41, 428.28, -13.47) mm, rotated rx 180 ry 0 rz -11.91 deg; joints [13.586, -29.453, 82.019, -88.351, 90.76, 141.715]
  MoveL 1774 to (-206.47, 428.01, -13.48) mm, rotated rx -180 ry 0 rz -11.91 deg; joints [13.586, -29.467, 82.051, -88.35, 90.76, 141.732]
  MoveL 1775 to (-206.5, 427.77, -13.47) mm, rotated rx -180 ry 0 rz -11.91 deg; joints [13.587, -29.48, 82.079, -88.349, 90.76, 141.747]
  MoveL 1776 to (-206.52, 427.53, -13.48) mm, rotated rx 180 ry 0 rz -11.91 deg; joints [13.589, -29.493, 82.106, -88.348, 90.76, 141.762]
  MoveL 1777 to (-206.52, 427.04, -13.48) mm, rotated rx -180 ry 0 rz -11.91 deg; joints [13.592, -29.518, 82.161, -88.345, 90.762, 141.792]
  MoveL 1778 to (-206.52, 50.21, -13.47) mm, rotated rx -180 ry 0 rz -11.91 deg; joints [17.408, -44.794, 117.193, -84.546, 91.309, 161.612]
  MoveL 1779 to (-206.51, 49.73, -13.47) mm, rotated rx -180 ry 0 rz -11.91 deg; joints [17.415, -44.809, 117.231, -84.539, 91.309, 161.635]
  MoveL 1780 to (-206.48, 49.48, -13.47) mm, rotated rx -180 ry 0 rz -11.91 deg; joints [17.42, -44.817, 117.25, -84.535, 91.309, 161.647]
  MoveL 1781 to (-206.43, 49.24, -13.47) mm, rotated rx 180 ry 0 rz -11.91 deg; joints [17.425, -44.824, 117.268, -84.53, 91.309, 161.657]
  MoveL 1782 to (-206.37, 49.02, -13.47) mm, rotated rx -180 ry 0 rz -11.91 deg; joints [17.43, -44.831, 117.284, -84.524, 91.31, 161.667]
  MoveL 1783 to (-206.28, 48.8, -13.48) mm, rotated rx -180 ry 0 rz -11.91 deg; joints [17.436, -44.837, 117.3, -84.518, 91.311, 161.677]
  MoveL 1784 to (-206.18, 48.57, -13.48) mm, rotated rx -180 ry 0 rz -11.91 deg; joints [17.443, -44.843, 117.315, -84.511, 91.312, 161.686]
  MoveL 1785 to (-206.06, 48.35, -13.48) mm, rotated rx -180 ry 0 rz -11.91 deg; joints [17.451, -44.849, 117.33, -84.504, 91.314, 161.695]
  MoveL 1786 to (-205.98, 48.22, -13.48) mm, rotated rx -180 ry 0 rz -11.91 deg; joints [17.456, -44.852, 117.338, -84.499, 91.315, 161.7]
  MoveL 1787 to (-205.88, 48.09, -13.48) mm, rotated rx -180 ry 0 rz -11.91 deg; joints [17.462, -44.856, 117.346, -84.493, 91.316, 161.705]
  MoveL 1788 to (-205.78, 47.96, -13.48) mm, rotated rx 180 ry 0 rz -11.91 deg; joints [17.468, -44.859, 117.354, -84.488, 91.317, 161.71]
  MoveL 1789 to (-205.66, 47.83, -13.48) mm, rotated rx -180 ry 0 rz -11.91 deg; joints [17.474, -44.862, 117.361, -84.481, 91.319, 161.714]
  MoveL 1790 to (-205.51, 47.67, -13.47) mm, rotated rx -180 ry 0 rz -11.91 deg; joints [17.483, -44.866, 117.37, -84.473, 91.321, 161.72]
  MoveL 1791 to (-205.35, 47.54, -13.48) mm, rotated rx 180 ry 0 rz -11.91 deg; joints [17.491, -44.868, 117.377, -84.465, 91.323, 161.724]
  MoveL 1792 to (-205.19, 47.42, -13.48) mm, rotated rx -180 ry 0 rz -11.91 deg; joints [17.499, -44.871, 117.383, -84.457, 91.325, 161.727]
  MoveL 1793 to (-205.03, 47.31, -13.48) mm, rotated rx 180 ry 0 rz -11.91 deg; joints [17.507, -44.873, 117.387, -84.45, 91.327, 161.73]
  MoveL 1794 to (-204.81, 47.18, -13.48) mm, rotated rx -180 ry 0 rz -11.91 deg; joints [17.518, -44.875, 117.392, -84.439, 91.33, 161.733]
  MoveL 1795 to (-204.58, 47.08, -13.48) mm, rotated rx -180 ry 0 rz -11.91 deg; joints [17.528, -44.876, 117.395, -84.429, 91.333, 161.735]
  MoveL 1796 to (-204.36, 46.99, -13.47) mm, rotated rx -180 ry 0 rz -11.91 deg; joints [17.538, -44.876, 117.396, -84.419, 91.336, 161.736]
  MoveL 1797 to (-204.13, 46.92, -13.47) mm, rotated rx -180 ry 0 rz -11.91 deg; joints [17.548, -44.876, 117.395, -84.41, 91.339, 161.736]
  MoveL 1798 to (-203.89, 46.87, -13.48) mm, rotated rx 180 ry 0 rz -11.91 deg; joints [17.559, -44.876, 117.393, -84.4, 91.343, 161.735]
  MoveL 1799 to (-203.65, 46.84, -13.47) mm, rotated rx -180 ry 0 rz -11.91 deg; joints [17.569, -44.874, 117.39, -84.39, 91.346, 161.733]
  MoveL 1800 to (-203.41, 46.83, -13.47) mm, rotated rx -180 ry 0 rz -11.91 deg; joints [17.579, -44.873, 117.385, -84.381, 91.349, 161.73]
  MoveL 1801 to (-203.17, 46.82, -13.48) mm, rotated rx 180 ry 0 rz -11.91 deg; joints [17.589, -44.87, 117.379, -84.371, 91.352, 161.727]
  MoveL 1802 to (222.09, 46.82, -13.48) mm, rotated rx 180 ry 0 rz -11.91 deg; joints [33.035, -38.227, 101.047, -70.77, 99.157, 153.581]
  MoveL 1803 to (223.29, 46.83, -13.48) mm, rotated rx 180 ry 0 rz -11.91 deg; joints [33.073, -38.2, 100.984, -70.741, 99.185, 153.552]
  MoveL 1804 to (223.53, 46.84, -13.47) mm, rotated rx 180 ry 0 rz -11.91 deg; joints [33.08, -38.194, 100.971, -70.736, 99.191, 153.546]
  MoveL 1805 to (223.77, 46.87, -13.48) mm, rotated rx -180 ry 0 rz -11.91 deg; joints [33.087, -38.188, 100.956, -70.731, 99.197, 153.539]
  MoveL 1806 to (224.01, 46.92, -13.48) mm, rotated rx -180 ry 0 rz -11.91 deg; joints [33.093, -38.181, 100.939, -70.726, 99.203, 153.531]
  MoveL 1807 to (224.24, 46.99, -13.47) mm, rotated rx 180 ry 0 rz -11.91 deg; joints [33.099, -38.173, 100.922, -70.722, 99.208, 153.522]
  MoveL 1808 to (224.46, 47.08, -13.47) mm, rotated rx -180 ry 0 rz -11.91 deg; joints [33.104, -38.165, 100.903, -70.719, 99.214, 153.513]
  MoveL 1809 to (224.69, 47.18, -13.47) mm, rotated rx -180 ry 0 rz -11.91 deg; joints [33.109, -38.157, 100.883, -70.716, 99.22, 153.503]
  MoveL 1810 to (224.92, 47.31, -13.48) mm, rotated rx -180 ry 0 rz -11.91 deg; joints [33.114, -38.147, 100.861, -70.714, 99.226, 153.492]
  MoveL 1811 to (225.07, 47.42, -13.47) mm, rotated rx -180 ry 0 rz -11.91 deg; joints [33.117, -38.14, 100.845, -70.713, 99.23, 153.483]
  MoveL 1812 to (225.23, 47.54, -13.48) mm, rotated rx 180 ry 0 rz -11.91 deg; joints [33.119, -38.132, 100.827, -70.712, 99.235, 153.474]
  MoveL 1813 to (225.39, 47.67, -13.48) mm, rotated rx -180 ry 0 rz -11.91 deg; joints [33.121, -38.124, 100.808, -70.712, 99.239, 153.464]
  MoveL 1814 to (225.55, 47.83, -13.48) mm, rotated rx 180 ry 0 rz -11.91 deg; joints [33.123, -38.115, 100.787, -70.712, 99.244, 153.453]
  MoveL 1815 to (225.66, 47.96, -13.48) mm, rotated rx 180 ry 0 rz -11.91 deg; joints [33.124, -38.108, 100.771, -70.713, 99.247, 153.444]
  MoveL 1816 to (225.77, 48.09, -13.47) mm, rotated rx -180 ry 0 rz -11.91 deg; joints [33.125, -38.101, 100.755, -70.714, 99.251, 153.436]
  MoveL 1817 to (225.86, 48.22, -13.47) mm, rotated rx 180 ry 0 rz -11.91 deg; joints [33.125, -38.094, 100.74, -70.715, 99.253, 153.428]
  MoveL 1818 to (225.94, 48.35, -13.47) mm, rotated rx 180 ry 0 rz -11.91 deg; joints [33.125, -38.088, 100.725, -70.716, 99.256, 153.42]
  MoveL 1819 to (226.07, 48.57, -13.48) mm, rotated rx -180 ry 0 rz -11.91 deg; joints [33.124, -38.077, 100.701, -70.719, 99.26, 153.407]
  MoveL 1820 to (226.17, 48.8, -13.48) mm, rotated rx -180 ry 0 rz -11.91 deg; joints [33.123, -38.067, 100.678, -70.722, 99.264, 153.394]
  MoveL 1821 to (226.25, 49.02, -13.48) mm, rotated rx -180 ry 0 rz -11.91 deg; joints [33.121, -38.058, 100.656, -70.726, 99.267, 153.382]
  MoveL 1822 to (226.31, 49.24, -13.48) mm, rotated rx 180 ry 0 rz -11.91 deg; joints [33.118, -38.048, 100.635, -70.73, 99.27, 153.37]
  MoveL 1823 to (226.36, 49.48, -13.48) mm, rotated rx -180 ry 0 rz -11.91 deg; joints [33.115, -38.039, 100.613, -70.735, 99.273, 153.358]
  MoveL 1824 to (226.39, 49.73, -13.48) mm, rotated rx 180 ry 0 rz -11.91 deg; joints [33.111, -38.03, 100.592, -70.741, 99.275, 153.346]
  MoveL 1825 to (226.4, 50.21, -13.48) mm, rotated rx -180 ry 0 rz -11.91 deg; joints [33.101, -38.012, 100.553, -70.753, 99.278, 153.324]
  MoveL 1826 to (226.4, 428.01, -13.48) mm, rotated rx 180 ry 0 rz -11.91 deg; joints [26.697, -20.377, 62.253, -79.643, 100.754, 132.037]
  MoveL 1827 to (226.4, 428.22, -13.48) mm, rotated rx -180 ry 0 rz -11.91 deg; joints [26.694, -20.363, 62.224, -79.648, 100.754, 132.022]
  MoveL 1828 to (226.38, 428.44, -13.48) mm, rotated rx 180 ry 0 rz -11.91 deg; joints [26.691, -20.349, 62.195, -79.653, 100.754, 132.006]
  MoveL 1829 to (226.35, 428.65, -13.48) mm, rotated rx -180 ry 0 rz -11.91 deg; joints [26.687, -20.336, 62.168, -79.658, 100.754, 131.991]
  MoveL 1830 to (226.3, 428.87, -13.47) mm, rotated rx -180 ry 0 rz -11.91 deg; joints [26.682, -20.324, 62.142, -79.664, 100.753, 131.977]
  MoveL 1831 to (226.24, 429.08, -13.48) mm, rotated rx 180 ry 0 rz -11.91 deg; joints [26.678, -20.312, 62.116, -79.67, 100.752, 131.963]
  MoveL 1832 to (226.16, 429.3, -13.48) mm, rotated rx -180 ry 0 rz -11.91 deg; joints [26.672, -20.3, 62.092, -79.676, 100.751, 131.95]
  MoveL 1833 to (226.06, 429.51, -13.48) mm, rotated rx -180 ry 0 rz -11.91 deg; joints [26.667, -20.289, 62.07, -79.682, 100.749, 131.937]
  MoveL 1834 to (225.94, 429.73, -13.48) mm, rotated rx -180 ry 0 rz -11.91 deg; joints [26.66, -20.279, 62.048, -79.688, 100.746, 131.925]
  MoveL 1835 to (225.8, 429.94, -13.48) mm, rotated rx -180 ry 0 rz -11.91 deg; joints [26.654, -20.27, 62.028, -79.695, 100.743, 131.914]
  MoveL 1836 to (225.6, 430.19, -13.47) mm, rotated rx -180 ry 0 rz -11.91 deg; joints [26.645, -20.26, 62.008, -79.703, 100.738, 131.902]
  MoveL 1837 to (225.35, 430.44, -13.48) mm, rotated rx -180 ry 0 rz -11.91 deg; joints [26.634, -20.252, 61.991, -79.712, 100.732, 131.892]
  MoveL 1838 to (225.13, 430.62, -13.48) mm, rotated rx -180 ry 0 rz -11.91 deg; joints [26.626, -20.247, 61.981, -79.719, 100.727, 131.885]
  MoveL 1839 to (224.91, 430.77, -13.47) mm, rotated rx -180 ry 0 rz -11.91 deg; joints [26.617, -20.244, 61.975, -79.725, 100.721, 131.881]
  MoveL 1840 to (224.68, 430.9, -13.47) mm, rotated rx -180 ry 0 rz -11.91 deg; joints [26.609, -20.243, 61.973, -79.731, 100.716, 131.879]
  MoveL 1841 to (224.46, 431, -13.48) mm, rotated rx -180 ry 0 rz -11.91 deg; joints [26.602, -20.244, 61.974, -79.736, 100.71, 131.879]
  MoveL 1842 to (224.24, 431.09, -13.47) mm, rotated rx -180 ry 0 rz -11.91 deg; joints [26.595, -20.245, 61.978, -79.741, 100.704, 131.88]
  MoveL 1843 to (224.01, 431.15, -13.48) mm, rotated rx -180 ry 0 rz -11.91 deg; joints [26.587, -20.248, 61.985, -79.745, 100.698, 131.883]
  MoveL 1844 to (223.77, 431.21, -13.47) mm, rotated rx 180 ry 0 rz -11.91 deg; joints [26.58, -20.253, 61.994, -79.749, 100.692, 131.887]
  MoveL 1845 to (223.53, 431.24, -13.48) mm, rotated rx 180 ry 0 rz -11.91 deg; joints [26.573, -20.258, 62.007, -79.753, 100.686, 131.892]
  MoveL 1846 to (223.29, 431.25, -13.48) mm, rotated rx -180 ry 0 rz -11.91 deg; joints [26.566, -20.265, 62.021, -79.756, 100.679, 131.899]
  MoveL 1847 to (223.05, 431.25, -13.47) mm, rotated rx -180 ry 0 rz -11.91 deg; joints [26.56, -20.273, 62.038, -79.759, 100.673, 131.907]
  MoveL 1848 to (-164.9, 431.25, -13.48) mm, rotated rx -180 ry 0 rz -11.91 deg; joints [14.909, -28.763, 80.489, -87.323, 91.603, 140.907]
  Set speed (38.1 mm/s)
  MoveL 1849 to (-165.25, 432.42, -13.48) mm, rotated rx 180 ry 0 rz -11.91 deg; joints [14.887, -28.706, 80.368, -87.342, 91.593, 140.841]
  MoveL 1850 to (-164.27, 433.07, -13.48) mm, rotated rx -180 ry 0 rz -11.91 deg; joints [14.913, -28.658, 80.263, -87.323, 91.611, 140.785]
  Set speed (25.4 mm/s)
  MoveL 1851 to (-164.27, 433.07, -15.84) mm, rotated rx 180 ry 0 rz -11.91 deg; joints [14.914, -28.548, 80.238, -87.32, 91.608, 140.87]
  MoveL 1852 to (-164.27, 432.44, -16.48) mm, rotated rx -180 ry 0 rz -11.91 deg; joints [14.92, -28.551, 80.303, -87.314, 91.608, 140.932]
  Set speed (38.1 mm/s)
  MoveL 1853 to (-164.9, 431.8, -16.48) mm, rotated rx 180 ry 0 rz -11.91 deg; joints [14.905, -28.593, 80.394, -87.324, 91.597, 140.981]
  Set speed (76.2 mm/s)
  MoveL 1854 to (-194.97, 431.8, -16.48) mm, rotated rx -180 ry 0 rz -11.91 deg; joints [13.931, -28.988, 81.274, -88.081, 90.979, 141.442]
  MoveL 1855 to (-199.31, 431.8, -16.48) mm, rotated rx 180 ry 0 rz -11.91 deg; joints [13.79, -29.042, 81.395, -88.192, 90.891, 141.506]
  MoveL 1856 to (-199.79, 431.8, -16.48) mm, rotated rx -180 ry 0 rz -11.91 deg; joints [13.775, -29.048, 81.409, -88.204, 90.881, 141.513]
  MoveL 1857 to (-200.03, 431.77, -16.47) mm, rotated rx 180 ry 0 rz -11.91 deg; joints [13.767, -29.052, 81.419, -88.21, 90.876, 141.518]
  MoveL 1858 to (-200.27, 431.73, -16.47) mm, rotated rx -180 ry 0 rz -11.91 deg; joints [13.76, -29.058, 81.43, -88.216, 90.871, 141.524]
  MoveL 1859 to (-200.52, 431.67, -16.47) mm, rotated rx -180 ry 0 rz -11.91 deg; joints [13.752, -29.064, 81.444, -88.222, 90.867, 141.532]
  MoveL 1860 to (-204.13, 430.52, -16.47) mm, rotated rx -180 ry 0 rz -11.91 deg; joints [13.643, -29.168, 81.672, -88.306, 90.797, 141.655]
  MoveL 1861 to (-204.42, 430.43, -16.48) mm, rotated rx 180 ry 0 rz -11.91 deg; joints [13.635, -29.176, 81.691, -88.313, 90.791, 141.665]
  MoveL 1862 to (-204.57, 430.37, -16.48) mm, rotated rx -180 ry 0 rz -11.91 deg; joints [13.63, -29.181, 81.702, -88.316, 90.788, 141.67]
  MoveL 1863 to (-204.72, 430.31, -16.48) mm, rotated rx -180 ry 0 rz -11.91 deg; joints [13.626, -29.186, 81.713, -88.319, 90.785, 141.676]
  MoveL 1864 to (-204.86, 430.23, -16.48) mm, rotated rx -180 ry 0 rz -11.91 deg; joints [13.622, -29.192, 81.725, -88.323, 90.783, 141.683]
  MoveL 1865 to (-205.01, 430.15, -16.48) mm, rotated rx -180 ry 0 rz -11.91 deg; joints [13.618, -29.198, 81.739, -88.326, 90.78, 141.69]
  MoveL 1866 to (-205.16, 430.05, -16.48) mm, rotated rx -180 ry 0 rz -11.91 deg; joints [13.614, -29.205, 81.754, -88.329, 90.777, 141.698]
  MoveL 1867 to (-205.3, 429.94, -16.47) mm, rotated rx -180 ry 0 rz -11.91 deg; joints [13.61, -29.212, 81.77, -88.332, 90.775, 141.707]
  MoveL 1868 to (-205.53, 429.75, -16.48) mm, rotated rx -180 ry 0 rz -11.91 deg; joints [13.604, -29.225, 81.798, -88.336, 90.771, 141.722]
  MoveL 1869 to (-205.75, 429.52, -16.48) mm, rotated rx 180 ry 0 rz -11.91 deg; joints [13.599, -29.239, 81.83, -88.34, 90.767, 141.739]
  MoveL 1870 to (-205.92, 429.3, -16.48) mm, rotated rx -180 ry 0 rz -11.91 deg; joints [13.595, -29.252, 81.859, -88.343, 90.764, 141.755]
  MoveL 1871 to (-206.06, 429.09, -16.48) mm, rotated rx -180 ry 0 rz -11.91 deg; joints [13.592, -29.265, 81.886, -88.345, 90.762, 141.77]
  MoveL 1872 to (-206.14, 428.95, -16.48) mm, rotated rx 180 ry 0 rz -11.91 deg; joints [13.59, -29.273, 81.904, -88.346, 90.761, 141.779]
  MoveL 1873 to (-206.21, 428.82, -16.47) mm, rotated rx -180 ry 0 rz -11.91 deg; joints [13.589, -29.281, 81.921, -88.347, 90.76, 141.789]
  MoveL 1874 to (-206.27, 428.69, -16.48) mm, rotated rx 180 ry 0 rz -11.91 deg; joints [13.588, -29.289, 81.937, -88.348, 90.759, 141.798]
  MoveL 1875 to (-206.32, 428.55, -16.48) mm, rotated rx -180 ry 0 rz -11.91 deg; joints [13.588, -29.296, 81.954, -88.348, 90.758, 141.807]
  MoveL 1876 to (-206.37, 428.42, -16.48) mm, rotated rx -180 ry 0 rz -11.91 deg; joints [13.587, -29.304, 81.97, -88.348, 90.758, 141.816]
  MoveL 1877 to (-206.41, 428.28, -16.47) mm, rotated rx -180 ry 0 rz -11.91 deg; joints [13.587, -29.311, 81.987, -88.349, 90.757, 141.824]
  MoveL 1878 to (-206.47, 428.01, -16.48) mm, rotated rx 180 ry 0 rz -11.91 deg; joints [13.587, -29.326, 82.019, -88.348, 90.757, 141.842]
  MoveL 1879 to (-206.5, 427.77, -16.48) mm, rotated rx -180 ry 0 rz -11.91 deg; joints [13.588, -29.339, 82.047, -88.347, 90.757, 141.857]
  MoveL 1880 to (-206.52, 427.53, -16.47) mm, rotated rx -180 ry 0 rz -11.91 deg; joints [13.589, -29.351, 82.074, -88.346, 90.757, 141.872]
  MoveL 1881 to (-206.52, 427.04, -16.47) mm, rotated rx 180 ry 0 rz -11.91 deg; joints [13.593, -29.376, 82.128, -88.343, 90.759, 141.901]
  MoveL 1882 to (-206.52, 50.21, -16.47) mm, rotated rx 180 ry 0 rz -11.91 deg; joints [17.41, -44.608, 117.161, -84.542, 91.294, 161.766]
  MoveL 1883 to (-206.51, 49.73, -16.48) mm, rotated rx 180 ry 0 rz -11.91 deg; joints [17.416, -44.623, 117.199, -84.535, 91.294, 161.789]
  MoveL 1884 to (-206.48, 49.48, -16.47) mm, rotated rx -180 ry 0 rz -11.91 deg; joints [17.421, -44.63, 117.218, -84.53, 91.295, 161.8]
  MoveL 1885 to (-206.43, 49.24, -16.47) mm, rotated rx -180 ry 0 rz -11.91 deg; joints [17.426, -44.638, 117.236, -84.525, 91.295, 161.811]
  MoveL 1886 to (-206.37, 49.02, -16.47) mm, rotated rx -180 ry 0 rz -11.91 deg; joints [17.431, -44.644, 117.252, -84.52, 91.296, 161.821]
  MoveL 1887 to (-206.28, 48.8, -16.48) mm, rotated rx 180 ry 0 rz -11.91 deg; joints [17.437, -44.65, 117.268, -84.514, 91.297, 161.831]
  MoveL 1888 to (-206.18, 48.57, -16.48) mm, rotated rx 180 ry 0 rz -11.91 deg; joints [17.444, -44.657, 117.283, -84.507, 91.298, 161.84]
  MoveL 1889 to (-206.06, 48.35, -16.48) mm, rotated rx -180 ry 0 rz -11.91 deg; joints [17.452, -44.663, 117.298, -84.499, 91.299, 161.849]
  MoveL 1890 to (-205.98, 48.22, -16.48) mm, rotated rx 180 ry 0 rz -11.91 deg; joints [17.457, -44.666, 117.306, -84.494, 91.3, 161.854]
  MoveL 1891 to (-205.88, 48.09, -16.47) mm, rotated rx 180 ry 0 rz -11.91 deg; joints [17.463, -44.669, 117.314, -84.489, 91.302, 161.859]
  MoveL 1892 to (-205.78, 47.96, -16.48) mm, rotated rx -180 ry 0 rz -11.91 deg; joints [17.469, -44.672, 117.322, -84.483, 91.303, 161.864]
  MoveL 1893 to (-205.66, 47.83, -16.48) mm, rotated rx 180 ry 0 rz -11.91 deg; joints [17.475, -44.675, 117.329, -84.477, 91.304, 161.868]
  MoveL 1894 to (-205.51, 47.67, -16.47) mm, rotated rx 180 ry 0 rz -11.91 deg; joints [17.484, -44.679, 117.338, -84.469, 91.306, 161.873]
  MoveL 1895 to (-205.35, 47.54, -16.48) mm, rotated rx -180 ry 0 rz -11.91 deg; joints [17.492, -44.682, 117.345, -84.461, 91.308, 161.878]
  MoveL 1896 to (-205.19, 47.42, -16.47) mm, rotated rx 180 ry 0 rz -11.91 deg; joints [17.5, -44.684, 117.351, -84.453, 91.31, 161.881]
  MoveL 1897 to (-205.03, 47.31, -16.47) mm, rotated rx -180 ry 0 rz -11.91 deg; joints [17.508, -44.686, 117.355, -84.445, 91.313, 161.884]
  MoveL 1898 to (-204.81, 47.18, -16.48) mm, rotated rx 180 ry 0 rz -11.91 deg; joints [17.519, -44.688, 117.36, -84.435, 91.316, 161.887]
  MoveL 1899 to (-204.58, 47.08, -16.48) mm, rotated rx -180 ry 0 rz -11.91 deg; joints [17.529, -44.689, 117.362, -84.425, 91.319, 161.889]
  MoveL 1900 to (-204.36, 46.99, -16.48) mm, rotated rx -180 ry 0 rz -11.91 deg; joints [17.54, -44.69, 117.364, -84.415, 91.322, 161.89]
  MoveL 1901 to (-204.13, 46.92, -16.47) mm, rotated rx -180 ry 0 rz -11.91 deg; joints [17.55, -44.69, 117.363, -84.405, 91.325, 161.89]
  MoveL 1902 to (-203.89, 46.87, -16.47) mm, rotated rx -180 ry 0 rz -11.91 deg; joints [17.56, -44.689, 117.361, -84.395, 91.328, 161.889]
  MoveL 1903 to (-203.65, 46.84, -16.48) mm, rotated rx 180 ry 0 rz -11.91 deg; joints [17.57, -44.688, 117.358, -84.385, 91.331, 161.887]
  MoveL 1904 to (-203.41, 46.83, -16.48) mm, rotated rx -180 ry 0 rz -11.91 deg; joints [17.58, -44.686, 117.353, -84.376, 91.334, 161.884]
  MoveL 1905 to (-203.17, 46.83, -16.47) mm, rotated rx -180 ry 0 rz -11.91 deg; joints [17.59, -44.684, 117.347, -84.367, 91.338, 161.881]
  MoveL 1906 to (222.09, 46.82, -16.48) mm, rotated rx 180 ry 0 rz -11.91 deg; joints [33.036, -38.067, 101.016, -70.75, 99.115, 153.705]
  MoveL 1907 to (223.29, 46.83, -16.48) mm, rotated rx -180 ry 0 rz -11.91 deg; joints [33.074, -38.04, 100.954, -70.72, 99.143, 153.676]
  MoveL 1908 to (223.53, 46.84, -16.47) mm, rotated rx -180 ry 0 rz -11.91 deg; joints [33.081, -38.035, 100.94, -70.715, 99.149, 153.67]
  MoveL 1909 to (223.77, 46.87, -16.47) mm, rotated rx -180 ry 0 rz -11.91 deg; joints [33.088, -38.028, 100.925, -70.71, 99.155, 153.663]
  MoveL 1910 to (224.01, 46.92, -16.48) mm, rotated rx 180 ry 0 rz -11.91 deg; joints [33.095, -38.021, 100.909, -70.705, 99.161, 153.654]
  MoveL 1911 to (224.24, 46.99, -16.47) mm, rotated rx -180 ry 0 rz -11.91 deg; joints [33.101, -38.014, 100.892, -70.701, 99.166, 153.646]
  MoveL 1912 to (224.46, 47.08, -16.48) mm, rotated rx -180 ry 0 rz -11.91 deg; joints [33.106, -38.006, 100.873, -70.698, 99.172, 153.637]
  MoveL 1913 to (224.69, 47.18, -16.47) mm, rotated rx -180 ry 0 rz -11.91 deg; joints [33.111, -37.997, 100.853, -70.695, 99.178, 153.627]
  MoveL 1914 to (224.92, 47.31, -16.48) mm, rotated rx -180 ry 0 rz -11.91 deg; joints [33.115, -37.988, 100.831, -70.693, 99.184, 153.615]
  MoveL 1915 to (225.07, 47.42, -16.47) mm, rotated rx -180 ry 0 rz -11.91 deg; joints [33.118, -37.98, 100.814, -70.692, 99.188, 153.607]
  MoveL 1916 to (225.23, 47.54, -16.47) mm, rotated rx -180 ry 0 rz -11.91 deg; joints [33.12, -37.973, 100.797, -70.691, 99.193, 153.597]
  MoveL 1917 to (225.39, 47.67, -16.48) mm, rotated rx -180 ry 0 rz -11.91 deg; joints [33.123, -37.964, 100.777, -70.691, 99.197, 153.587]
  MoveL 1918 to (225.55, 47.83, -16.47) mm, rotated rx -180 ry 0 rz -11.91 deg; joints [33.124, -37.955, 100.757, -70.691, 99.202, 153.576]
  MoveL 1919 to (225.66, 47.96, -16.48) mm, rotated rx 180 ry 0 rz -11.91 deg; joints [33.125, -37.948, 100.74, -70.692, 99.205, 153.568]
  MoveL 1920 to (225.77, 48.09, -16.48) mm, rotated rx 180 ry 0 rz -11.91 deg; joints [33.126, -37.941, 100.724, -70.693, 99.209, 153.559]
  MoveL 1921 to (225.86, 48.22, -16.48) mm, rotated rx 180 ry 0 rz -11.91 deg; joints [33.126, -37.935, 100.709, -70.694, 99.211, 153.551]
  MoveL 1922 to (225.94, 48.35, -16.47) mm, rotated rx -180 ry 0 rz -11.91 deg; joints [33.126, -37.928, 100.695, -70.695, 99.214, 153.543]
  MoveL 1923 to (226.07, 48.57, -16.48) mm, rotated rx 180 ry 0 rz -11.91 deg; joints [33.125, -37.918, 100.67, -70.698, 99.218, 153.53]
  MoveL 1924 to (226.17, 48.8, -16.48) mm, rotated rx -180 ry 0 rz -11.91 deg; joints [33.124, -37.908, 100.647, -70.701, 99.222, 153.517]
  MoveL 1925 to (226.25, 49.02, -16.47) mm, rotated rx -180 ry 0 rz -11.91 deg; joints [33.122, -37.898, 100.625, -70.705, 99.225, 153.505]
  MoveL 1926 to (226.31, 49.24, -16.47) mm, rotated rx -180 ry 0 rz -11.91 deg; joints [33.119, -37.889, 100.604, -70.709, 99.228, 153.493]
  MoveL 1927 to (226.36, 49.48, -16.47) mm, rotated rx 180 ry 0 rz -11.91 deg; joints [33.116, -37.879, 100.582, -70.714, 99.231, 153.481]
  MoveL 1928 to (226.39, 49.73, -16.48) mm, rotated rx -180 ry 0 rz -11.91 deg; joints [33.112, -37.87, 100.561, -70.72, 99.233, 153.469]
  MoveL 1929 to (226.4, 50.21, -16.47) mm, rotated rx -180 ry 0 rz -11.91 deg; joints [33.102, -37.853, 100.522, -70.732, 99.236, 153.447]
  MoveL 1930 to (226.4, 428.49, -16.47) mm, rotated rx -180 ry 0 rz -11.91 deg; joints [26.691, -20.213, 62.148, -79.636, 100.739, 132.096]
  MoveL 1931 to (226.4, 428.74, -16.47) mm, rotated rx -180 ry 0 rz -11.91 deg; joints [26.688, -20.197, 62.115, -79.642, 100.74, 132.078]
  MoveL 1932 to (226.38, 428.98, -16.47) mm, rotated rx -180 ry 0 rz -11.91 deg; joints [26.684, -20.182, 62.082, -79.647, 100.74, 132.06]
  MoveL 1933 to (226.35, 429.22, -16.48) mm, rotated rx 180 ry 0 rz -11.91 deg; joints [26.68, -20.167, 62.052, -79.653, 100.74, 132.043]
  MoveL 1934 to (226.29, 429.46, -16.47) mm, rotated rx -180 ry 0 rz -11.91 deg; joints [26.675, -20.153, 62.022, -79.66, 100.739, 132.027]
  MoveL 1935 to (226.22, 429.7, -16.48) mm, rotated rx -180 ry 0 rz -11.91 deg; joints [26.669, -20.14, 61.994, -79.666, 100.737, 132.012]
  MoveL 1936 to (226.12, 429.94, -16.47) mm, rotated rx -180 ry 0 rz -11.91 deg; joints [26.663, -20.127, 61.967, -79.673, 100.735, 131.997]
  MoveL 1937 to (226.04, 430.11, -16.47) mm, rotated rx 180 ry 0 rz -11.91 deg; joints [26.659, -20.119, 61.95, -79.678, 100.734, 131.987]
  MoveL 1938 to (225.94, 430.28, -16.47) mm, rotated rx 180 ry 0 rz -11.91 deg; joints [26.654, -20.111, 61.934, -79.683, 100.732, 131.978]
  MoveL 1939 to (225.86, 430.4, -16.47) mm, rotated rx -180 ry 0 rz -11.91 deg; joints [26.65, -20.105, 61.922, -79.687, 100.73, 131.971]
  MoveL 1940 to (225.77, 430.53, -16.48) mm, rotated rx -180 ry 0 rz -11.91 deg; joints [26.646, -20.1, 61.911, -79.691, 100.728, 131.965]
  MoveL 1941 to (225.68, 430.65, -16.48) mm, rotated rx 180 ry 0 rz -11.91 deg; joints [26.641, -20.095, 61.9, -79.695, 100.726, 131.959]
  MoveL 1942 to (225.57, 430.78, -16.48) mm, rotated rx 180 ry 0 rz -11.91 deg; joints [26.637, -20.09, 61.89, -79.699, 100.723, 131.953]
  MoveL 1943 to (225.42, 430.93, -16.48) mm, rotated rx -180 ry 0 rz -11.91 deg; joints [26.63, -20.085, 61.88, -79.704, 100.72, 131.947]
  MoveL 1944 to (225.27, 431.06, -16.48) mm, rotated rx -180 ry 0 rz -11.91 deg; joints [26.625, -20.081, 61.872, -79.709, 100.716, 131.942]
  MoveL 1945 to (225.12, 431.17, -16.48) mm, rotated rx -180 ry 0 rz -11.91 deg; joints [26.619, -20.078, 61.866, -79.714, 100.712, 131.938]
  MoveL 1946 to (224.98, 431.28, -16.48) mm, rotated rx -180 ry 0 rz -11.91 deg; joints [26.613, -20.076, 61.862, -79.718, 100.709, 131.935]
  MoveL 1947 to (224.74, 431.42, -16.47) mm, rotated rx 180 ry 0 rz -11.91 deg; joints [26.605, -20.075, 61.859, -79.724, 100.703, 131.932]
  MoveL 1948 to (224.5, 431.54, -16.48) mm, rotated rx -180 ry 0 rz -11.91 deg; joints [26.596, -20.075, 61.859, -79.73, 100.696, 131.932]
  MoveL 1949 to (224.25, 431.63, -16.47) mm, rotated rx -180 ry 0 rz -11.91 deg; joints [26.589, -20.077, 61.863, -79.735, 100.69, 131.933]
  MoveL 1950 to (224.01, 431.7, -16.48) mm, rotated rx -180 ry 0 rz -11.91 deg; joints [26.581, -20.08, 61.87, -79.739, 100.684, 131.935]
  MoveL 1951 to (223.77, 431.76, -16.48) mm, rotated rx -180 ry 0 rz -11.91 deg; joints [26.573, -20.084, 61.879, -79.744, 100.678, 131.939]
  MoveL 1952 to (223.53, 431.79, -16.47) mm, rotated rx -180 ry 0 rz -11.91 deg; joints [26.566, -20.09, 61.892, -79.747, 100.671, 131.945]
  MoveL 1953 to (223.29, 431.8, -16.48) mm, rotated rx -180 ry 0 rz -11.91 deg; joints [26.56, -20.097, 61.906, -79.751, 100.665, 131.952]
  MoveL 1954 to (223.05, 431.8, -16.48) mm, rotated rx -180 ry 0 rz -11.91 deg; joints [26.553, -20.105, 61.923, -79.753, 100.658, 131.96]
  MoveL 1955 to (-164.9, 431.8, -16.48) mm, rotated rx 180 ry 0 rz -11.91 deg; joints [14.905, -28.593, 80.394, -87.324, 91.597, 140.981]
  MoveL 1956 to (-194.97, 431.99, -17.53) mm, rotated rx 180 ry 0 rz -11.91 deg; joints [13.93, -28.928, 81.241, -88.082, 90.978, 141.468]
  MoveL 1957 to (-195.47, 431.99, -17.53) mm, rotated rx 180 ry 0 rz -11.91 deg; joints [13.914, -28.934, 81.255, -88.094, 90.967, 141.475]
  MoveL 1958 to (-198.35, 431.99, -17.52) mm, rotated rx -180 ry 0 rz -11.91 deg; joints [13.82, -28.97, 81.335, -88.168, 90.909, 141.518]
  MoveL 1959 to (-199.1, 431.99, -17.52) mm, rotated rx -180 ry 0 rz -11.91 deg; joints [13.796, -28.98, 81.356, -88.187, 90.894, 141.529]
  MoveL 1960 to (-199.28, 431.98, -17.53) mm, rotated rx 180 ry 0 rz -11.91 deg; joints [13.79, -28.983, 81.363, -88.192, 90.89, 141.532]
  MoveL 1961 to (-199.47, 431.96, -17.53) mm, rotated rx 180 ry 0 rz -11.91 deg; joints [13.784, -28.986, 81.371, -88.196, 90.886, 141.537]
  MoveL 1962 to (-199.66, 431.92, -17.53) mm, rotated rx -180 ry 0 rz -11.91 deg; joints [13.778, -28.991, 81.38, -88.201, 90.882, 141.542]
  MoveL 1963 to (-199.85, 431.88, -17.53) mm, rotated rx -180 ry 0 rz -11.91 deg; joints [13.772, -28.995, 81.39, -88.205, 90.879, 141.547]
  MoveL 1964 to (-200.27, 431.74, -17.52) mm, rotated rx -180 ry 0 rz -11.91 deg; joints [13.76, -29.007, 81.417, -88.215, 90.87, 141.562]
  MoveL 1965 to (-204.13, 430.52, -17.53) mm, rotated rx -180 ry 0 rz -11.91 deg; joints [13.644, -29.118, 81.661, -88.305, 90.796, 141.693]
  MoveL 1966 to (-204.42, 430.43, -17.53) mm, rotated rx 180 ry 0 rz -11.91 deg; joints [13.635, -29.127, 81.68, -88.312, 90.79, 141.703]
  MoveL 1967 to (-204.57, 430.37, -17.53) mm, rotated rx 180 ry 0 rz -11.91 deg; joints [13.631, -29.131, 81.69, -88.315, 90.787, 141.708]
  MoveL 1968 to (-204.72, 430.31, -17.52) mm, rotated rx -180 ry 0 rz -11.91 deg; joints [13.626, -29.137, 81.701, -88.319, 90.785, 141.714]
  MoveL 1969 to (-204.86, 430.23, -17.53) mm, rotated rx 180 ry 0 rz -11.91 deg; joints [13.622, -29.142, 81.714, -88.322, 90.782, 141.721]
  MoveL 1970 to (-205.01, 430.15, -17.53) mm, rotated rx -180 ry 0 rz -11.91 deg; joints [13.618, -29.148, 81.727, -88.325, 90.779, 141.728]
  MoveL 1971 to (-205.16, 430.05, -17.53) mm, rotated rx -180 ry 0 rz -11.91 deg; joints [13.614, -29.155, 81.742, -88.328, 90.776, 141.736]
  MoveL 1972 to (-205.3, 429.94, -17.52) mm, rotated rx -180 ry 0 rz -11.91 deg; joints [13.61, -29.162, 81.758, -88.331, 90.774, 141.745]
  MoveL 1973 to (-205.53, 429.75, -17.53) mm, rotated rx -180 ry 0 rz -11.91 deg; joints [13.604, -29.175, 81.786, -88.336, 90.77, 141.76]
  MoveL 1974 to (-205.75, 429.52, -17.52) mm, rotated rx -180 ry 0 rz -11.91 deg; joints [13.599, -29.19, 81.818, -88.34, 90.766, 141.778]
  MoveL 1975 to (-205.92, 429.3, -17.53) mm, rotated rx -180 ry 0 rz -11.91 deg; joints [13.595, -29.203, 81.847, -88.342, 90.763, 141.793]
  MoveL 1976 to (-206.06, 429.09, -17.52) mm, rotated rx -180 ry 0 rz -11.91 deg; joints [13.592, -29.216, 81.875, -88.345, 90.761, 141.808]
  MoveL 1977 to (-206.14, 428.95, -17.52) mm, rotated rx -180 ry 0 rz -11.91 deg; joints [13.591, -29.223, 81.892, -88.346, 90.76, 141.817]
  MoveL 1978 to (-206.21, 428.82, -17.53) mm, rotated rx -180 ry 0 rz -11.91 deg; joints [13.59, -29.231, 81.909, -88.346, 90.759, 141.827]
  MoveL 1979 to (-206.27, 428.69, -17.52) mm, rotated rx -180 ry 0 rz -11.91 deg; joints [13.589, -29.239, 81.926, -88.347, 90.758, 141.836]
  MoveL 1980 to (-206.32, 428.55, -17.52) mm, rotated rx -180 ry 0 rz -11.91 deg; joints [13.588, -29.247, 81.943, -88.348, 90.757, 141.845]
  MoveL 1981 to (-206.37, 428.42, -17.53) mm, rotated rx 180 ry 0 rz -11.91 deg; joints [13.587, -29.254, 81.959, -88.348, 90.757, 141.854]
  MoveL 1982 to (-206.41, 428.28, -17.53) mm, rotated rx 180 ry 0 rz -11.91 deg; joints [13.587, -29.261, 81.975, -88.348, 90.756, 141.862]
  MoveL 1983 to (-206.47, 428.01, -17.52) mm, rotated rx -180 ry 0 rz -11.91 deg; joints [13.587, -29.276, 82.007, -88.348, 90.756, 141.88]
  MoveL 1984 to (-206.5, 427.77, -17.53) mm, rotated rx 180 ry 0 rz -11.91 deg; joints [13.588, -29.289, 82.035, -88.347, 90.756, 141.895]
  MoveL 1985 to (-206.52, 427.53, -17.53) mm, rotated rx -180 ry 0 rz -11.91 deg; joints [13.59, -29.301, 82.063, -88.345, 90.757, 141.91]
  MoveL 1986 to (-206.52, 427.04, -17.53) mm, rotated rx 180 ry 0 rz -11.91 deg; joints [13.593, -29.326, 82.117, -88.342, 90.758, 141.939]
  MoveL 1987 to (-206.52, 50.21, -17.53) mm, rotated rx 180 ry 0 rz -11.91 deg; joints [17.41, -44.542, 117.149, -84.54, 91.289, 161.819]
  MoveL 1988 to (-206.51, 49.73, -17.53) mm, rotated rx -180 ry 0 rz -11.91 deg; joints [17.417, -44.558, 117.188, -84.533, 91.289, 161.843]
  MoveL 1989 to (-206.48, 49.48, -17.52) mm, rotated rx -180 ry 0 rz -11.91 deg; joints [17.421, -44.565, 117.206, -84.529, 91.289, 161.854]
  MoveL 1990 to (-206.43, 49.24, -17.53) mm, rotated rx 180 ry 0 rz -11.91 deg; joints [17.426, -44.572, 117.224, -84.524, 91.29, 161.865]
  MoveL 1991 to (-206.37, 49.02, -17.52) mm, rotated rx 180 ry 0 rz -11.91 deg; joints [17.432, -44.579, 117.241, -84.518, 91.291, 161.875]
  MoveL 1992 to (-206.28, 48.8, -17.52) mm, rotated rx -180 ry 0 rz -11.91 deg; joints [17.438, -44.585, 117.256, -84.512, 91.292, 161.884]
  MoveL 1993 to (-206.18, 48.57, -17.53) mm, rotated rx -180 ry 0 rz -11.91 deg; joints [17.445, -44.591, 117.272, -84.505, 91.293, 161.893]
  MoveL 1994 to (-206.06, 48.35, -17.52) mm, rotated rx -180 ry 0 rz -11.91 deg; joints [17.453, -44.597, 117.286, -84.497, 91.294, 161.902]
  MoveL 1995 to (-205.98, 48.22, -17.52) mm, rotated rx -180 ry 0 rz -11.91 deg; joints [17.458, -44.601, 117.295, -84.492, 91.295, 161.908]
  MoveL 1996 to (-205.88, 48.09, -17.53) mm, rotated rx -180 ry 0 rz -11.91 deg; joints [17.463, -44.604, 117.303, -84.487, 91.297, 161.912]
  MoveL 1997 to (-205.78, 47.96, -17.53) mm, rotated rx 180 ry 0 rz -11.91 deg; joints [17.469, -44.607, 117.31, -84.481, 91.298, 161.917]
  MoveL 1998 to (-205.66, 47.83, -17.52) mm, rotated rx -180 ry 0 rz -11.91 deg; joints [17.476, -44.61, 117.318, -84.475, 91.299, 161.922]
  MoveL 1999 to (-205.51, 47.67, -17.52) mm, rotated rx 180 ry 0 rz -11.91 deg; joints [17.484, -44.614, 117.327, -84.467, 91.301, 161.927]
  MoveL 2000 to (-205.35, 47.54, -17.53) mm, rotated rx -180 ry 0 rz -11.91 deg; joints [17.492, -44.617, 117.334, -84.459, 91.303, 161.932]
  MoveL 2001 to (-205.19, 47.42, -17.52) mm, rotated rx -180 ry 0 rz -11.91 deg; joints [17.5, -44.619, 117.339, -84.451, 91.305, 161.935]
  MoveL 2002 to (-205.03, 47.31, -17.53) mm, rotated rx 180 ry 0 rz -11.91 deg; joints [17.508, -44.621, 117.344, -84.444, 91.307, 161.938]
  MoveL 2003 to (-204.81, 47.18, -17.53) mm, rotated rx -180 ry 0 rz -11.91 deg; joints [17.519, -44.623, 117.348, -84.433, 91.31, 161.941]
  MoveL 2004 to (-204.58, 47.08, -17.53) mm, rotated rx 180 ry 0 rz -11.91 deg; joints [17.53, -44.624, 117.351, -84.423, 91.313, 161.943]
  MoveL 2005 to (-204.36, 46.99, -17.52) mm, rotated rx -180 ry 0 rz -11.91 deg; joints [17.54, -44.624, 117.352, -84.413, 91.316, 161.944]
  MoveL 2006 to (-204.13, 46.92, -17.53) mm, rotated rx -180 ry 0 rz -11.91 deg; joints [17.55, -44.624, 117.352, -84.404, 91.319, 161.943]
  MoveL 2007 to (-203.89, 46.87, -17.52) mm, rotated rx -180 ry 0 rz -11.91 deg; joints [17.56, -44.624, 117.35, -84.394, 91.323, 161.942]
  MoveL 2008 to (-203.65, 46.84, -17.52) mm, rotated rx -180 ry 0 rz -11.91 deg; joints [17.571, -44.622, 117.346, -84.384, 91.326, 161.941]
  MoveL 2009 to (-203.41, 46.83, -17.53) mm, rotated rx 180 ry 0 rz -11.91 deg; joints [17.581, -44.621, 117.341, -84.374, 91.329, 161.938]
  MoveL 2010 to (-203.17, 46.83, -17.53) mm, rotated rx -180 ry 0 rz -11.91 deg; joints [17.591, -44.618, 117.335, -84.365, 91.332, 161.934]
  MoveL 2011 to (222.09, 46.82, -17.52) mm, rotated rx -180 ry 0 rz -11.91 deg; joints [33.036, -38.011, 101.006, -70.742, 99.1, 153.748]
  MoveL 2012 to (223.29, 46.83, -17.52) mm, rotated rx -180 ry 0 rz -11.91 deg; joints [33.074, -37.984, 100.943, -70.713, 99.128, 153.719]
  MoveL 2013 to (223.53, 46.84, -17.53) mm, rotated rx 180 ry 0 rz -11.91 deg; joints [33.082, -37.979, 100.929, -70.707, 99.134, 153.713]
  MoveL 2014 to (223.77, 46.87, -17.53) mm, rotated rx 180 ry 0 rz -11.91 deg; joints [33.089, -37.972, 100.914, -70.702, 99.14, 153.706]
  MoveL 2015 to (224.01, 46.92, -17.53) mm, rotated rx -180 ry 0 rz -11.91 deg; joints [33.095, -37.965, 100.898, -70.698, 99.146, 153.698]
  MoveL 2016 to (224.24, 46.99, -17.53) mm, rotated rx 180 ry 0 rz -11.91 deg; joints [33.101, -37.958, 100.881, -70.694, 99.152, 153.689]
  MoveL 2017 to (224.46, 47.08, -17.52) mm, rotated rx -180 ry 0 rz -11.91 deg; joints [33.106, -37.95, 100.862, -70.691, 99.157, 153.68]
  MoveL 2018 to (224.69, 47.18, -17.53) mm, rotated rx 180 ry 0 rz -11.91 deg; joints [33.111, -37.941, 100.842, -70.688, 99.163, 153.67]
  MoveL 2019 to (224.92, 47.31, -17.53) mm, rotated rx -180 ry 0 rz -11.91 deg; joints [33.116, -37.932, 100.82, -70.686, 99.169, 153.659]
  MoveL 2020 to (225.07, 47.42, -17.53) mm, rotated rx -180 ry 0 rz -11.91 deg; joints [33.118, -37.925, 100.804, -70.685, 99.174, 153.65]
  MoveL 2021 to (225.23, 47.54, -17.52) mm, rotated rx -180 ry 0 rz -11.91 deg; joints [33.121, -37.917, 100.786, -70.684, 99.178, 153.641]
  MoveL 2022 to (225.39, 47.67, -17.52) mm, rotated rx -180 ry 0 rz -11.91 deg; joints [33.123, -37.909, 100.767, -70.684, 99.183, 153.631]
  MoveL 2023 to (225.55, 47.83, -17.52) mm, rotated rx 180 ry 0 rz -11.91 deg; joints [33.125, -37.9, 100.746, -70.684, 99.187, 153.62]
  MoveL 2024 to (225.66, 47.96, -17.52) mm, rotated rx -180 ry 0 rz -11.91 deg; joints [33.126, -37.892, 100.729, -70.685, 99.191, 153.611]
  MoveL 2025 to (225.77, 48.09, -17.53) mm, rotated rx -180 ry 0 rz -11.91 deg; joints [33.126, -37.886, 100.714, -70.685, 99.194, 153.602]
  MoveL 2026 to (225.86, 48.22, -17.53) mm, rotated rx -180 ry 0 rz -11.91 deg; joints [33.127, -37.879, 100.698, -70.687, 99.197, 153.594]
  MoveL 2027 to (225.94, 48.35, -17.53) mm, rotated rx -180 ry 0 rz -11.91 deg; joints [33.127, -37.873, 100.684, -70.688, 99.199, 153.586]
  MoveL 2028 to (226.07, 48.57, -17.53) mm, rotated rx -180 ry 0 rz -11.91 deg; joints [33.126, -37.862, 100.66, -70.691, 99.204, 153.573]
  MoveL 2029 to (226.17, 48.8, -17.52) mm, rotated rx -180 ry 0 rz -11.91 deg; joints [33.124, -37.852, 100.636, -70.694, 99.207, 153.561]
  MoveL 2030 to (226.25, 49.02, -17.53) mm, rotated rx 180 ry 0 rz -11.91 deg; joints [33.122, -37.842, 100.614, -70.698, 99.211, 153.548]
  MoveL 2031 to (226.31, 49.24, -17.53) mm, rotated rx -180 ry 0 rz -11.91 deg; joints [33.12, -37.833, 100.593, -70.702, 99.213, 153.537]
  MoveL 2032 to (226.36, 49.48, -17.53) mm, rotated rx -180 ry 0 rz -11.91 deg; joints [33.116, -37.824, 100.572, -70.707, 99.216, 153.524]
  MoveL 2033 to (226.39, 49.73, -17.53) mm, rotated rx 180 ry 0 rz -11.91 deg; joints [33.112, -37.815, 100.551, -70.712, 99.218, 153.512]
  MoveL 2034 to (226.4, 50.21, -17.52) mm, rotated rx -180 ry 0 rz -11.91 deg; joints [33.103, -37.797, 100.511, -70.724, 99.221, 153.49]
  MoveL 2035 to (226.4, 428.01, -17.53) mm, rotated rx 180 ry 0 rz -11.91 deg; joints [26.698, -20.198, 62.201, -79.618, 100.732, 132.164]
  MoveL 2036 to (226.4, 428.98, -17.52) mm, rotated rx -180 ry 0 rz -11.91 deg; joints [26.685, -20.135, 62.068, -79.641, 100.735, 132.092]
  MoveL 2037 to (226.38, 429.22, -17.53) mm, rotated rx -180 ry 0 rz -11.91 deg; joints [26.681, -20.12, 62.036, -79.647, 100.735, 132.075]
  MoveL 2038 to (226.34, 429.46, -17.52) mm, rotated rx -180 ry 0 rz -11.91 deg; joints [26.676, -20.105, 62.005, -79.653, 100.734, 132.058]
  MoveL 2039 to (226.28, 429.7, -17.52) mm, rotated rx -180 ry 0 rz -11.91 deg; joints [26.671, -20.091, 61.976, -79.659, 100.733, 132.042]
  MoveL 2040 to (226.2, 429.94, -17.53) mm, rotated rx -180 ry 0 rz -11.91 deg; joints [26.666, -20.078, 61.948, -79.666, 100.732, 132.027]
  MoveL 2041 to (226.15, 430.07, -17.53) mm, rotated rx 180 ry 0 rz -11.91 deg; joints [26.663, -20.071, 61.933, -79.669, 100.731, 132.019]
